ABB RAPID module: P708.mod

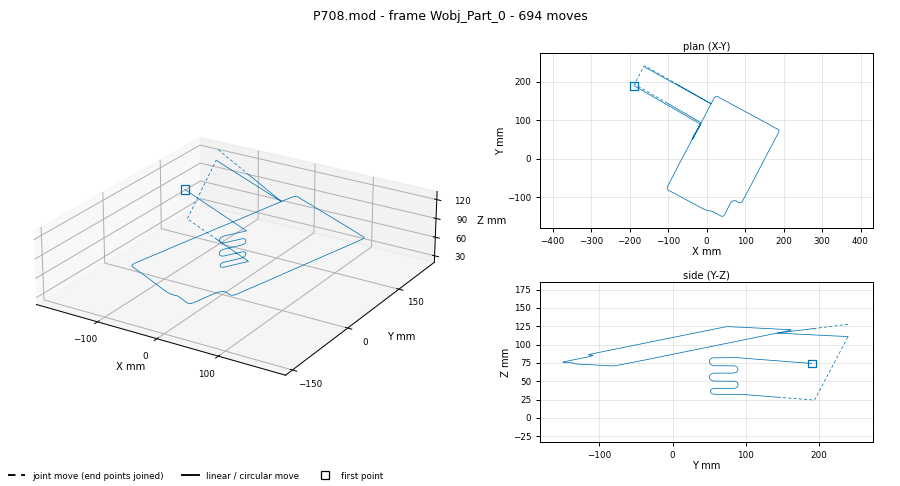
[picture p0: tool path of P708.mod in frame Wobj_Part_0, 694 of 704 moves have a stored position in this frame; points joined in program order, loops and branches not executed]
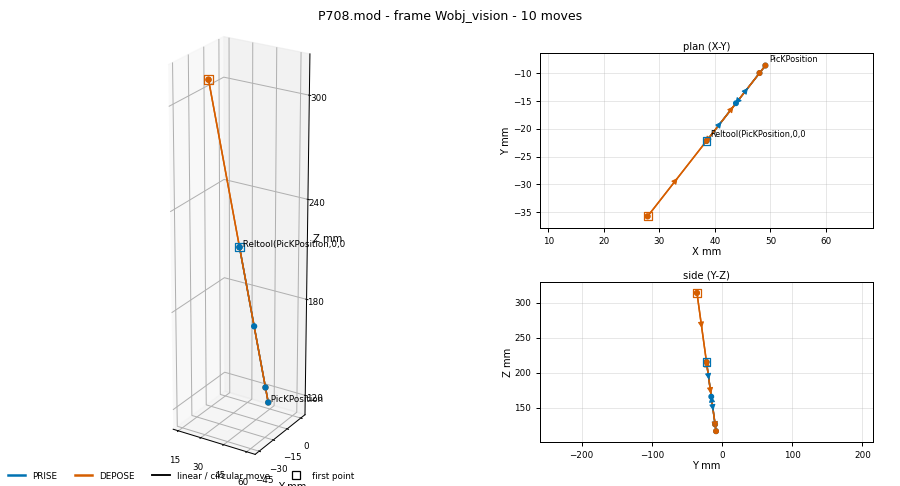
[picture p1: tool path of P708.mod in frame Wobj_vision, 10 of 704 moves have a stored position in this frame; points joined in program order, loops and branches not executed]
MODULE P708

    ! Nom         :P708
    ! Description :
    ! Créé le     :31/05/2023 18:09:45

    LOCAL CONST SPEEDDATA VitesseLente :=[3,500,0,0];
	LOCAL CONST SPEEDDATA VitesseRapide :=[30,500,0,0];
	LOCAL CONST SPEEDDATA VitesseTronconnage :=[2,500,0,0];
	LOCAL CONST SPEEDDATA VitesseTronconnageApp :=[10,500,0,0];
    !
    !Point de prise
    LOCAL PERS Robtarget PicKPosition := [[49.097436543476,-8.59484692597384,116.899947760068],[0.0805571048843757,-0.506621283374927,0.857813762365557,0.0316382234083716],[0,0,0,0],[8.999999E+09,8.999999E+09,8.999999E+09,8.999999E+09,8.999999E+09,8.999999E+09]];
	LOCAL PERS Pose Ref := [[0,0,0],[1,0,0,0]];
    !
    !Declaration des points de meulage

    !Tr_meulage_motif_1 : Meulage d'un motif
    LOCAL CONST Robtarget Tr_meulage_motif_1_0 := [[-15.398982421875,89.8560390625,82.14859375],[0.360190468749215,-0.346276211408762,0.600337290207395,-0.624460366733596],[0,0,0,0],[8.999999E+09,8.999999E+09,8.999999E+09,8.999999E+09,8.999999E+09,8.999999E+09]];
    LOCAL CONST Robtarget Tr_meulage_motif_1_1 := [[-15.875765625,88.977015625,82.148578125],[0.360190468749215,-0.346276211408762,0.600337290207395,-0.624460366733596],[0,0,0,0],[8.999999E+09,8.999999E+09,8.999999E+09,8.999999E+09,8.999999E+09,8.999999E+09]];
    LOCAL CONST Robtarget Tr_meulage_motif_1_2 := [[-16.352548828125,88.0979921875,82.1485625],[0.360190468749215,-0.346276211408762,0.600337290207395,-0.624460366733596],[0,0,0,0],[8.999999E+09,8.999999E+09,8.999999E+09,8.999999E+09,8.999999E+09,8.999999E+09]];
    LOCAL CONST Robtarget Tr_meulage_motif_1_3 := [[-16.82933203125,87.2189765625,82.148546875],[0.360190468749215,-0.346276211408762,0.600337290207395,-0.624460366733596],[0,0,0,0],[8.999999E+09,8.999999E+09,8.999999E+09,8.999999E+09,8.999999E+09,8.999999E+09]];
    LOCAL CONST Robtarget Tr_meulage_motif_1_4 := [[-17.306115234375,86.339953125,82.14853125],[0.360190468749215,-0.346276211408762,0.600337290207395,-0.624460366733596],[0,0,0,0],[8.999999E+09,8.999999E+09,8.999999E+09,8.999999E+09,8.999999E+09,8.999999E+09]];
    LOCAL CONST Robtarget Tr_meulage_motif_1_5 := [[-17.7828984375,85.4609296875,82.1485078125],[0.360190468749215,-0.346276211408762,0.600337290207395,-0.624460366733596],[0,0,0,0],[8.999999E+09,8.999999E+09,8.999999E+09,8.999999E+09,8.999999E+09,8.999999E+09]];
    LOCAL CONST Robtarget Tr_meulage_motif_1_6 := [[-18.259681640625,84.5819140625,82.1484921875],[0.360190468749215,-0.346276211408762,0.600337290207395,-0.624460366733596],[0,0,0,0],[8.999999E+09,8.999999E+09,8.999999E+09,8.999999E+09,8.999999E+09,8.999999E+09]];
    LOCAL CONST Robtarget Tr_meulage_motif_1_7 := [[-18.736462890625,83.702890625,82.1484765625],[0.360190468749215,-0.346276211408762,0.600337290207395,-0.624460366733596],[0,0,0,0],[8.999999E+09,8.999999E+09,8.999999E+09,8.999999E+09,8.999999E+09,8.999999E+09]];
    LOCAL CONST Robtarget Tr_meulage_motif_1_8 := [[-19.21324609375,82.8238671875,82.1484609375],[0.360190468749215,-0.346276211408762,0.600337290207395,-0.624460366733596],[0,0,0,0],[8.999999E+09,8.999999E+09,8.999999E+09,8.999999E+09,8.999999E+09,8.999999E+09]];
    LOCAL CONST Robtarget Tr_meulage_motif_1_9 := [[-19.690029296875,81.9448515625,82.1484453125],[0.360190468749215,-0.346276211408762,0.600337290207395,-0.624460366733596],[0,0,0,0],[8.999999E+09,8.999999E+09,8.999999E+09,8.999999E+09,8.999999E+09,8.999999E+09]];
    LOCAL CONST Robtarget Tr_meulage_motif_1_10 := [[-20.1668125,81.065828125,82.1484296875],[0.360190468749215,-0.346276211408762,0.600337290207395,-0.624460366733596],[0,0,0,0],[8.999999E+09,8.999999E+09,8.999999E+09,8.999999E+09,8.999999E+09,8.999999E+09]];
    LOCAL CONST Robtarget Tr_meulage_motif_1_11 := [[-20.643595703125,80.1868046875,82.1484140625],[0.360190468749215,-0.346276211408762,0.600337290207395,-0.624460366733596],[0,0,0,0],[8.999999E+09,8.999999E+09,8.999999E+09,8.999999E+09,8.999999E+09,8.999999E+09]];
    LOCAL CONST Robtarget Tr_meulage_motif_1_12 := [[-21.12037890625,79.3077890625,82.1483984375],[0.360190468749215,-0.346276211408762,0.600337290207395,-0.624460366733596],[0,0,0,0],[8.999999E+09,8.999999E+09,8.999999E+09,8.999999E+09,8.999999E+09,8.999999E+09]];
    LOCAL CONST Robtarget Tr_meulage_motif_1_13 := [[-21.597162109375,78.428765625,82.1483828125],[0.360190468749215,-0.346276211408762,0.600337290207395,-0.624460366733596],[0,0,0,0],[8.999999E+09,8.999999E+09,8.999999E+09,8.999999E+09,8.999999E+09,8.999999E+09]];
    LOCAL CONST Robtarget Tr_meulage_motif_1_14 := [[-22.0739453125,77.5497421875,82.1483671875],[0.360190468749215,-0.346276211408762,0.600337290207395,-0.624460366733596],[0,0,0,0],[8.999999E+09,8.999999E+09,8.999999E+09,8.999999E+09,8.999999E+09,8.999999E+09]];
    LOCAL CONST Robtarget Tr_meulage_motif_1_15 := [[-22.550728515625,76.6707265625,82.1483515625],[0.360190468749215,-0.346276211408762,0.600337290207395,-0.624460366733596],[0,0,0,0],[8.999999E+09,8.999999E+09,8.999999E+09,8.999999E+09,8.999999E+09,8.999999E+09]];
    LOCAL CONST Robtarget Tr_meulage_motif_1_16 := [[-23.02751171875,75.791703125,82.1483359375],[0.360190468749215,-0.346276211408762,0.600337290207395,-0.624460366733596],[0,0,0,0],[8.999999E+09,8.999999E+09,8.999999E+09,8.999999E+09,8.999999E+09,8.999999E+09]];
    LOCAL CONST Robtarget Tr_meulage_motif_1_17 := [[-23.504294921875,74.9126796875,82.1483203125],[0.360190468749215,-0.346276211408762,0.600337290207395,-0.624460366733596],[0,0,0,0],[8.999999E+09,8.999999E+09,8.999999E+09,8.999999E+09,8.999999E+09,8.999999E+09]];
    LOCAL CONST Robtarget Tr_meulage_motif_1_18 := [[-23.981078125,74.03365625,82.1483046875],[0.360190468749215,-0.346276211408762,0.600337290207395,-0.624460366733596],[0,0,0,0],[8.999999E+09,8.999999E+09,8.999999E+09,8.999999E+09,8.999999E+09,8.999999E+09]];
    LOCAL CONST Robtarget Tr_meulage_motif_1_19 := [[-24.457861328125,73.154640625,82.1482890625],[0.360190468749215,-0.346276211408762,0.600337290207395,-0.624460366733596],[0,0,0,0],[8.999999E+09,8.999999E+09,8.999999E+09,8.999999E+09,8.999999E+09,8.999999E+09]];
    LOCAL CONST Robtarget Tr_meulage_motif_1_20 := [[-24.93464453125,72.2756171875,82.1482734375],[0.360190468749215,-0.346276211408762,0.600337290207395,-0.624460366733596],[0,0,0,0],[8.999999E+09,8.999999E+09,8.999999E+09,8.999999E+09,8.999999E+09,8.999999E+09]];
    LOCAL CONST Robtarget Tr_meulage_motif_1_21 := [[-25.411427734375,71.39659375,82.1482578125],[0.360190468749215,-0.346276211408762,0.600337290207395,-0.624460366733596],[0,0,0,0],[8.999999E+09,8.999999E+09,8.999999E+09,8.999999E+09,8.999999E+09,8.999999E+09]];
    LOCAL CONST Robtarget Tr_meulage_motif_1_22 := [[-25.888208984375,70.517578125,82.1482421875],[0.360190468749215,-0.346276211408762,0.600337290207395,-0.624460366733596],[0,0,0,0],[8.999999E+09,8.999999E+09,8.999999E+09,8.999999E+09,8.999999E+09,8.999999E+09]];
    LOCAL CONST Robtarget Tr_meulage_motif_1_23 := [[-26.3649921875,69.6385546875,82.14821875],[0.360190468749215,-0.346276211408762,0.600337290207395,-0.624460366733596],[0,0,0,0],[8.999999E+09,8.999999E+09,8.999999E+09,8.999999E+09,8.999999E+09,8.999999E+09]];
    LOCAL CONST Robtarget Tr_meulage_motif_1_24 := [[-26.841775390625,68.75953125,82.148203125],[0.360190468749215,-0.346276211408762,0.600337290207395,-0.624460366733596],[0,0,0,0],[8.999999E+09,8.999999E+09,8.999999E+09,8.999999E+09,8.999999E+09,8.999999E+09]];
    LOCAL CONST Robtarget Tr_meulage_motif_1_25 := [[-27.31855859375,67.880515625,82.1481875],[0.360190468749215,-0.346276211408762,0.600337290207395,-0.624460366733596],[0,0,0,0],[8.999999E+09,8.999999E+09,8.999999E+09,8.999999E+09,8.999999E+09,8.999999E+09]];
    LOCAL CONST Robtarget Tr_meulage_motif_1_26 := [[-27.795341796875,67.0014921875,82.148171875],[0.360190468749215,-0.346276211408762,0.600337290207395,-0.624460366733596],[0,0,0,0],[8.999999E+09,8.999999E+09,8.999999E+09,8.999999E+09,8.999999E+09,8.999999E+09]];
    LOCAL CONST Robtarget Tr_meulage_motif_1_27 := [[-28.272125,66.12246875,82.14815625],[0.360190468749215,-0.346276211408762,0.600337290207395,-0.624460366733596],[0,0,0,0],[8.999999E+09,8.999999E+09,8.999999E+09,8.999999E+09,8.999999E+09,8.999999E+09]];
    LOCAL CONST Robtarget Tr_meulage_motif_1_28 := [[-28.748908203125,65.24344921875,82.148140625],[0.360190468749215,-0.346276211408762,0.600337290207395,-0.624460366733596],[0,0,0,0],[8.999999E+09,8.999999E+09,8.999999E+09,8.999999E+09,8.999999E+09,8.999999E+09]];
    LOCAL CONST Robtarget Tr_meulage_motif_1_29 := [[-29.22569140625,64.3644296875,82.148125],[0.360190468749215,-0.346276211408762,0.600337290207395,-0.624460366733596],[0,0,0,0],[8.999999E+09,8.999999E+09,8.999999E+09,8.999999E+09,8.999999E+09,8.999999E+09]];
    LOCAL CONST Robtarget Tr_meulage_motif_1_30 := [[-29.702474609375,63.48540625,82.148109375],[0.360190468749215,-0.346276211408762,0.600337290207395,-0.624460366733596],[0,0,0,0],[8.999999E+09,8.999999E+09,8.999999E+09,8.999999E+09,8.999999E+09,8.999999E+09]];
    LOCAL CONST Robtarget Tr_meulage_motif_1_31 := [[-30.1792578125,62.60638671875,82.14809375],[0.360190468749215,-0.346276211408762,0.600337290207395,-0.624460366733596],[0,0,0,0],[8.999999E+09,8.999999E+09,8.999999E+09,8.999999E+09,8.999999E+09,8.999999E+09]];
    LOCAL CONST Robtarget Tr_meulage_motif_1_32 := [[-30.656041015625,61.7273671875,82.148078125],[0.360190468749215,-0.346276211408762,0.600337290207395,-0.624460366733596],[0,0,0,0],[8.999999E+09,8.999999E+09,8.999999E+09,8.999999E+09,8.999999E+09,8.999999E+09]];
    LOCAL CONST Robtarget Tr_meulage_motif_1_33 := [[-31.13282421875,60.84834375,82.1480625],[0.360190468749215,-0.346276211408762,0.600337290207395,-0.624460366733596],[0,0,0,0],[8.999999E+09,8.999999E+09,8.999999E+09,8.999999E+09,8.999999E+09,8.999999E+09]];
    LOCAL CONST Robtarget Tr_meulage_motif_1_34 := [[-31.609607421875,59.96932421875,82.148046875],[0.360190468749215,-0.346276211408762,0.600337290207395,-0.624460366733596],[0,0,0,0],[8.999999E+09,8.999999E+09,8.999999E+09,8.999999E+09,8.999999E+09,8.999999E+09]];
    LOCAL CONST Robtarget Tr_meulage_motif_1_35 := [[-32.086390625,59.0903046875,82.14803125],[0.360190468749215,-0.346276211408762,0.600337290207395,-0.624460366733596],[0,0,0,0],[8.999999E+09,8.999999E+09,8.999999E+09,8.999999E+09,8.999999E+09,8.999999E+09]];
    LOCAL CONST Robtarget Tr_meulage_motif_1_36 := [[-32.563173828125,58.21128125,82.148015625],[0.360190468749215,-0.346276211408762,0.600337290207395,-0.624460366733596],[0,0,0,0],[8.999999E+09,8.999999E+09,8.999999E+09,8.999999E+09,8.999999E+09,8.999999E+09]];
    LOCAL CONST Robtarget Tr_meulage_motif_1_37 := [[-33.03995703125,57.33226171875,82.148],[0.360190468749215,-0.346276211408762,0.600337290207395,-0.624460366733596],[0,0,0,0],[8.999999E+09,8.999999E+09,8.999999E+09,8.999999E+09,8.999999E+09,8.999999E+09]];
    LOCAL CONST Robtarget Tr_meulage_motif_1_38 := [[-33.51673828125,56.45323828125,82.147984375],[0.360190468749215,-0.346276211408762,0.600337290207395,-0.624460366733596],[0,0,0,0],[8.999999E+09,8.999999E+09,8.999999E+09,8.999999E+09,8.999999E+09,8.999999E+09]];
    LOCAL CONST Robtarget Tr_meulage_motif_1_39 := [[-33.9913828125,55.58151953125,82.0373828125],[0.360190468749215,-0.346276211408762,0.600337290207395,-0.624460366733596],[0,0,0,0],[8.999999E+09,8.999999E+09,8.999999E+09,8.999999E+09,8.999999E+09,8.999999E+09]];
    LOCAL CONST Robtarget Tr_meulage_motif_1_40 := [[-34.44533984375,54.75098828125,81.826203125],[0.360190468749215,-0.346276211408762,0.600337290207395,-0.624460366733596],[0,0,0,0],[8.999999E+09,8.999999E+09,8.999999E+09,8.999999E+09,8.999999E+09,8.999999E+09]];
    LOCAL CONST Robtarget Tr_meulage_motif_1_41 := [[-34.855359375,54.00330859375,81.554375],[0.360190468749215,-0.346276211408762,0.600337290207395,-0.624460366733596],[0,0,0,0],[8.999999E+09,8.999999E+09,8.999999E+09,8.999999E+09,8.999999E+09,8.999999E+09]];
    LOCAL CONST Robtarget Tr_meulage_motif_1_42 := [[-35.216421875,53.34600390625,81.278453125],[0.360190468749215,-0.346276211408762,0.600337290207395,-0.624460366733596],[0,0,0,0],[8.999999E+09,8.999999E+09,8.999999E+09,8.999999E+09,8.999999E+09,8.999999E+09]];
    LOCAL CONST Robtarget Tr_meulage_motif_1_43 := [[-35.74921875,52.38240625,80.662375],[0.360190468749215,-0.346276211408762,0.600337290207395,-0.624460366733596],[0,0,0,0],[8.999999E+09,8.999999E+09,8.999999E+09,8.999999E+09,8.999999E+09,8.999999E+09]];
    LOCAL CONST Robtarget Tr_meulage_motif_1_44 := [[-36.24816015625,51.4882578125,79.8147890625],[0.360190468749215,-0.346276211408762,0.600337290207395,-0.624460366733596],[0,0,0,0],[8.999999E+09,8.999999E+09,8.999999E+09,8.999999E+09,8.999999E+09,8.999999E+09]];
    LOCAL CONST Robtarget Tr_meulage_motif_1_45 := [[-36.6653203125,50.7502265625,78.7910078125],[0.360190468749215,-0.346276211408762,0.600337290207395,-0.624460366733596],[0,0,0,0],[8.999999E+09,8.999999E+09,8.999999E+09,8.999999E+09,8.999999E+09,8.999999E+09]];
    LOCAL CONST Robtarget Tr_meulage_motif_1_46 := [[-36.91225,50.32884375,77.6749296875],[0.360190468749215,-0.346276211408762,0.600337290207395,-0.624460366733596],[0,0,0,0],[8.999999E+09,8.999999E+09,8.999999E+09,8.999999E+09,8.999999E+09,8.999999E+09]];
    LOCAL CONST Robtarget Tr_meulage_motif_1_47 := [[-36.934,50.30986328125,76.97903125],[0.360190468749215,-0.346276211408762,0.600337290207395,-0.624460366733596],[0,0,0,0],[8.999999E+09,8.999999E+09,8.999999E+09,8.999999E+09,8.999999E+09,8.999999E+09]];
    LOCAL CONST Robtarget Tr_meulage_motif_1_48 := [[-36.94240234375,50.31443359375,76.3178515625],[0.360190468749215,-0.346276211408762,0.600337290207395,-0.624460366733596],[0,0,0,0],[8.999999E+09,8.999999E+09,8.999999E+09,8.999999E+09,8.999999E+09,8.999999E+09]];
    LOCAL CONST Robtarget Tr_meulage_motif_1_49 := [[-36.924640625,50.3672421875,75.656828125],[0.360190468749215,-0.346276211408762,0.600337290207395,-0.624460366733596],[0,0,0,0],[8.999999E+09,8.999999E+09,8.999999E+09,8.999999E+09,8.999999E+09,8.999999E+09]];
    LOCAL CONST Robtarget Tr_meulage_motif_1_50 := [[-36.7011015625,50.81280078125,74.555203125],[0.360190468749215,-0.346276211408762,0.600337290207395,-0.624460366733596],[0,0,0,0],[8.999999E+09,8.999999E+09,8.999999E+09,8.999999E+09,8.999999E+09,8.999999E+09]];
    LOCAL CONST Robtarget Tr_meulage_motif_1_51 := [[-36.30547265625,51.57275,73.5486953125],[0.360190468749215,-0.346276211408762,0.600337290207395,-0.624460366733596],[0,0,0,0],[8.999999E+09,8.999999E+09,8.999999E+09,8.999999E+09,8.999999E+09,8.999999E+09]];
    LOCAL CONST Robtarget Tr_meulage_motif_1_52 := [[-35.8280625,52.47807421875,72.7199296875],[0.360190468749215,-0.346276211408762,0.600337290207395,-0.624460366733596],[0,0,0,0],[8.999999E+09,8.999999E+09,8.999999E+09,8.999999E+09,8.999999E+09,8.999999E+09]];
    LOCAL CONST Robtarget Tr_meulage_motif_1_53 := [[-35.5055,53.08477734375,72.3242265625],[0.360190468749215,-0.346276211408762,0.600337290207395,-0.624460366733596],[0,0,0,0],[8.999999E+09,8.999999E+09,8.999999E+09,8.999999E+09,8.999999E+09,8.999999E+09]];
    LOCAL CONST Robtarget Tr_meulage_motif_1_54 := [[-34.95950390625,54.10619140625,71.836765625],[0.360190468749215,-0.346276211408762,0.600337290207395,-0.624460366733596],[0,0,0,0],[8.999999E+09,8.999999E+09,8.999999E+09,8.999999E+09,8.999999E+09,8.999999E+09]];
    LOCAL CONST Robtarget Tr_meulage_motif_1_55 := [[-34.55996484375,54.85081640625,71.5727109375],[0.360190468749215,-0.346276211408762,0.600337290207395,-0.624460366733596],[0,0,0,0],[8.999999E+09,8.999999E+09,8.999999E+09,8.999999E+09,8.999999E+09,8.999999E+09]];
    LOCAL CONST Robtarget Tr_meulage_motif_1_56 := [[-34.118203125,55.67148046875,71.36828125],[0.360190468749215,-0.346276211408762,0.600337290207395,-0.624460366733596],[0,0,0,0],[8.999999E+09,8.999999E+09,8.999999E+09,8.999999E+09,8.999999E+09,8.999999E+09]];
    LOCAL CONST Robtarget Tr_meulage_motif_1_57 := [[-33.65158984375,56.53504296875,71.25971875],[0.360190468749215,-0.346276211408762,0.600337290207395,-0.624460366733596],[0,0,0,0],[8.999999E+09,8.999999E+09,8.999999E+09,8.999999E+09,8.999999E+09,8.999999E+09]];
    LOCAL CONST Robtarget Tr_meulage_motif_1_58 := [[-33.1797578125,57.40829296875,71.1491484375],[0.360190468749215,-0.346276211408762,0.600337290207395,-0.624460366733596],[0,0,0,0],[8.999999E+09,8.999999E+09,8.999999E+09,8.999999E+09,8.999999E+09,8.999999E+09]];
    LOCAL CONST Robtarget Tr_meulage_motif_1_59 := [[-32.702974609375,58.2873125,71.1491640625],[0.360190468749215,-0.346276211408762,0.600337290207395,-0.624460366733596],[0,0,0,0],[8.999999E+09,8.999999E+09,8.999999E+09,8.999999E+09,8.999999E+09,8.999999E+09]];
    LOCAL CONST Robtarget Tr_meulage_motif_1_60 := [[-32.22619140625,59.16633203125,71.1491796875],[0.360190468749215,-0.346276211408762,0.600337290207395,-0.624460366733596],[0,0,0,0],[8.999999E+09,8.999999E+09,8.999999E+09,8.999999E+09,8.999999E+09,8.999999E+09]];
    LOCAL CONST Robtarget Tr_meulage_motif_1_61 := [[-31.74941015625,60.04535546875,71.1491953125],[0.360190468749215,-0.346276211408762,0.600337290207395,-0.624460366733596],[0,0,0,0],[8.999999E+09,8.999999E+09,8.999999E+09,8.999999E+09,8.999999E+09,8.999999E+09]];
    LOCAL CONST Robtarget Tr_meulage_motif_1_62 := [[-31.272626953125,60.924375,71.1492109375],[0.360190468749215,-0.346276211408762,0.600337290207395,-0.624460366733596],[0,0,0,0],[8.999999E+09,8.999999E+09,8.999999E+09,8.999999E+09,8.999999E+09,8.999999E+09]];
    LOCAL CONST Robtarget Tr_meulage_motif_1_63 := [[-30.79584375,61.80339453125,71.1492265625],[0.360190468749215,-0.346276211408762,0.600337290207395,-0.624460366733596],[0,0,0,0],[8.999999E+09,8.999999E+09,8.999999E+09,8.999999E+09,8.999999E+09,8.999999E+09]];
    LOCAL CONST Robtarget Tr_meulage_motif_1_64 := [[-30.319060546875,62.68241796875,71.1492421875],[0.360190468749215,-0.346276211408762,0.600337290207395,-0.624460366733596],[0,0,0,0],[8.999999E+09,8.999999E+09,8.999999E+09,8.999999E+09,8.999999E+09,8.999999E+09]];
    LOCAL CONST Robtarget Tr_meulage_motif_1_65 := [[-29.84227734375,63.5614375,71.1492578125],[0.360190468749215,-0.346276211408762,0.600337290207395,-0.624460366733596],[0,0,0,0],[8.999999E+09,8.999999E+09,8.999999E+09,8.999999E+09,8.999999E+09,8.999999E+09]];
    LOCAL CONST Robtarget Tr_meulage_motif_1_66 := [[-29.365494140625,64.4404609375,71.14928125],[0.360190468749215,-0.346276211408762,0.600337290207395,-0.624460366733596],[0,0,0,0],[8.999999E+09,8.999999E+09,8.999999E+09,8.999999E+09,8.999999E+09,8.999999E+09]];
    LOCAL CONST Robtarget Tr_meulage_motif_1_67 := [[-28.8887109375,65.31948046875,71.149296875],[0.360190468749215,-0.346276211408762,0.600337290207395,-0.624460366733596],[0,0,0,0],[8.999999E+09,8.999999E+09,8.999999E+09,8.999999E+09,8.999999E+09,8.999999E+09]];
    LOCAL CONST Robtarget Tr_meulage_motif_1_68 := [[-28.411927734375,66.1985,71.1493125],[0.360190468749215,-0.346276211408762,0.600337290207395,-0.624460366733596],[0,0,0,0],[8.999999E+09,8.999999E+09,8.999999E+09,8.999999E+09,8.999999E+09,8.999999E+09]];
    LOCAL CONST Robtarget Tr_meulage_motif_1_69 := [[-27.93514453125,67.0775234375,71.149328125],[0.360190468749215,-0.346276211408762,0.600337290207395,-0.624460366733596],[0,0,0,0],[8.999999E+09,8.999999E+09,8.999999E+09,8.999999E+09,8.999999E+09,8.999999E+09]];
    LOCAL CONST Robtarget Tr_meulage_motif_1_70 := [[-27.458361328125,67.956546875,71.14934375],[0.360190468749215,-0.346276211408762,0.600337290207395,-0.624460366733596],[0,0,0,0],[8.999999E+09,8.999999E+09,8.999999E+09,8.999999E+09,8.999999E+09,8.999999E+09]];
    LOCAL CONST Robtarget Tr_meulage_motif_1_71 := [[-26.981578125,68.8355625,71.149359375],[0.360190468749215,-0.346276211408762,0.600337290207395,-0.624460366733596],[0,0,0,0],[8.999999E+09,8.999999E+09,8.999999E+09,8.999999E+09,8.999999E+09,8.999999E+09]];
    LOCAL CONST Robtarget Tr_meulage_motif_1_72 := [[-26.504794921875,69.7145859375,71.149375],[0.360190468749215,-0.346276211408762,0.600337290207395,-0.624460366733596],[0,0,0,0],[8.999999E+09,8.999999E+09,8.999999E+09,8.999999E+09,8.999999E+09,8.999999E+09]];
    LOCAL CONST Robtarget Tr_meulage_motif_1_73 := [[-26.02801171875,70.593609375,71.149390625],[0.360190468749215,-0.346276211408762,0.600337290207395,-0.624460366733596],[0,0,0,0],[8.999999E+09,8.999999E+09,8.999999E+09,8.999999E+09,8.999999E+09,8.999999E+09]];
    LOCAL CONST Robtarget Tr_meulage_motif_1_74 := [[-25.551228515625,71.472625,71.14940625],[0.360190468749215,-0.346276211408762,0.600337290207395,-0.624460366733596],[0,0,0,0],[8.999999E+09,8.999999E+09,8.999999E+09,8.999999E+09,8.999999E+09,8.999999E+09]];
    LOCAL CONST Robtarget Tr_meulage_motif_1_75 := [[-25.0744453125,72.3516484375,71.149421875],[0.360190468749215,-0.346276211408762,0.600337290207395,-0.624460366733596],[0,0,0,0],[8.999999E+09,8.999999E+09,8.999999E+09,8.999999E+09,8.999999E+09,8.999999E+09]];
    LOCAL CONST Robtarget Tr_meulage_motif_1_76 := [[-24.5976640625,73.230671875,71.1494375],[0.360190468749215,-0.346276211408762,0.600337290207395,-0.624460366733596],[0,0,0,0],[8.999999E+09,8.999999E+09,8.999999E+09,8.999999E+09,8.999999E+09,8.999999E+09]];
    LOCAL CONST Robtarget Tr_meulage_motif_1_77 := [[-24.120880859375,74.1096875,71.149453125],[0.360190468749215,-0.346276211408762,0.600337290207395,-0.624460366733596],[0,0,0,0],[8.999999E+09,8.999999E+09,8.999999E+09,8.999999E+09,8.999999E+09,8.999999E+09]];
    LOCAL CONST Robtarget Tr_meulage_motif_1_78 := [[-23.64409765625,74.9887109375,71.14946875],[0.360190468749215,-0.346276211408762,0.600337290207395,-0.624460366733596],[0,0,0,0],[8.999999E+09,8.999999E+09,8.999999E+09,8.999999E+09,8.999999E+09,8.999999E+09]];
    LOCAL CONST Robtarget Tr_meulage_motif_1_79 := [[-23.167314453125,75.867734375,71.149484375],[0.360190468749215,-0.346276211408762,0.600337290207395,-0.624460366733596],[0,0,0,0],[8.999999E+09,8.999999E+09,8.999999E+09,8.999999E+09,8.999999E+09,8.999999E+09]];
    LOCAL CONST Robtarget Tr_meulage_motif_1_80 := [[-22.69053125,76.74675,71.1495],[0.360190468749215,-0.346276211408762,0.600337290207395,-0.624460366733596],[0,0,0,0],[8.999999E+09,8.999999E+09,8.999999E+09,8.999999E+09,8.999999E+09,8.999999E+09]];
    LOCAL CONST Robtarget Tr_meulage_motif_1_81 := [[-22.213748046875,77.6257734375,71.149515625],[0.360190468749215,-0.346276211408762,0.600337290207395,-0.624460366733596],[0,0,0,0],[8.999999E+09,8.999999E+09,8.999999E+09,8.999999E+09,8.999999E+09,8.999999E+09]];
    LOCAL CONST Robtarget Tr_meulage_motif_1_82 := [[-21.73696484375,78.504796875,71.14953125],[0.360190468749215,-0.346276211408762,0.600337290207395,-0.624460366733596],[0,0,0,0],[8.999999E+09,8.999999E+09,8.999999E+09,8.999999E+09,8.999999E+09,8.999999E+09]];
    LOCAL CONST Robtarget Tr_meulage_motif_1_83 := [[-21.260181640625,79.3838125,71.149546875],[0.360190468749215,-0.346276211408762,0.600337290207395,-0.624460366733596],[0,0,0,0],[8.999999E+09,8.999999E+09,8.999999E+09,8.999999E+09,8.999999E+09,8.999999E+09]];
    LOCAL CONST Robtarget Tr_meulage_motif_1_84 := [[-20.7833984375,80.2628359375,71.1495703125],[0.360190468749215,-0.346276211408762,0.600337290207395,-0.624460366733596],[0,0,0,0],[8.999999E+09,8.999999E+09,8.999999E+09,8.999999E+09,8.999999E+09,8.999999E+09]];
    LOCAL CONST Robtarget Tr_meulage_motif_1_85 := [[-20.306615234375,81.141859375,71.1495859375],[0.360190468749215,-0.346276211408762,0.600337290207395,-0.624460366733596],[0,0,0,0],[8.999999E+09,8.999999E+09,8.999999E+09,8.999999E+09,8.999999E+09,8.999999E+09]];
    LOCAL CONST Robtarget Tr_meulage_motif_1_86 := [[-19.82983203125,82.020875,71.1496015625],[0.360190468749215,-0.346276211408762,0.600337290207395,-0.624460366733596],[0,0,0,0],[8.999999E+09,8.999999E+09,8.999999E+09,8.999999E+09,8.999999E+09,8.999999E+09]];
    LOCAL CONST Robtarget Tr_meulage_motif_1_87 := [[-19.353048828125,82.8998984375,71.1496171875],[0.360190468749215,-0.346276211408762,0.600337290207395,-0.624460366733596],[0,0,0,0],[8.999999E+09,8.999999E+09,8.999999E+09,8.999999E+09,8.999999E+09,8.999999E+09]];
    LOCAL CONST Robtarget Tr_meulage_motif_1_88 := [[-18.876265625,83.778921875,71.1496328125],[0.360190468749215,-0.346276211408762,0.600337290207395,-0.624460366733596],[0,0,0,0],[8.999999E+09,8.999999E+09,8.999999E+09,8.999999E+09,8.999999E+09,8.999999E+09]];
    LOCAL CONST Robtarget Tr_meulage_motif_1_89 := [[-18.404435546875,84.652171875,71.0390625],[0.360190468749215,-0.346276211408762,0.600337290207395,-0.624460366733596],[0,0,0,0],[8.999999E+09,8.999999E+09,8.999999E+09,8.999999E+09,8.999999E+09,8.999999E+09]];
    LOCAL CONST Robtarget Tr_meulage_motif_1_90 := [[-17.95584375,85.485625,70.8279140625],[0.360190468749215,-0.346276211408762,0.600337290207395,-0.624460366733596],[0,0,0,0],[8.999999E+09,8.999999E+09,8.999999E+09,8.999999E+09,8.999999E+09,8.999999E+09]];
    LOCAL CONST Robtarget Tr_meulage_motif_1_91 := [[-17.552736328125,86.2370546875,70.556109375],[0.360190468749215,-0.346276211408762,0.600337290207395,-0.624460366733596],[0,0,0,0],[8.999999E+09,8.999999E+09,8.999999E+09,8.999999E+09,8.999999E+09,8.999999E+09]];
    LOCAL CONST Robtarget Tr_meulage_motif_1_92 := [[-17.21737109375,86.8645859375,70.252],[0.360190468749215,-0.346276211408762,0.600337290207395,-0.624460366733596],[0,0,0,0],[8.999999E+09,8.999999E+09,8.999999E+09,8.999999E+09,8.999999E+09,8.999999E+09]];
    LOCAL CONST Robtarget Tr_meulage_motif_1_93 := [[-16.73257421875,87.778484375,69.5895546875],[0.360190468749215,-0.346276211408762,0.600337290207395,-0.624460366733596],[0,0,0,0],[8.999999E+09,8.999999E+09,8.999999E+09,8.999999E+09,8.999999E+09,8.999999E+09]];
    LOCAL CONST Robtarget Tr_meulage_motif_1_94 := [[-16.3140087890625,88.5775390625,68.6877265625],[0.360190468749215,-0.346276211408762,0.600337290207395,-0.624460366733596],[0,0,0,0],[8.999999E+09,8.999999E+09,8.999999E+09,8.999999E+09,8.999999E+09,8.999999E+09]];
    LOCAL CONST Robtarget Tr_meulage_motif_1_95 := [[-16.0722392578125,89.055015625,67.6418125],[0.360190468749215,-0.346276211408762,0.600337290207395,-0.624460366733596],[0,0,0,0],[8.999999E+09,8.999999E+09,8.999999E+09,8.999999E+09,8.999999E+09,8.999999E+09]];
    LOCAL CONST Robtarget Tr_meulage_motif_1_96 := [[-15.99294921875,89.222234375,66.948671875],[0.360190468749215,-0.346276211408762,0.600337290207395,-0.624460366733596],[0,0,0,0],[8.999999E+09,8.999999E+09,8.999999E+09,8.999999E+09,8.999999E+09,8.999999E+09]];
    LOCAL CONST Robtarget Tr_meulage_motif_1_97 := [[-15.9722958984375,89.2836796875,66.17875],[0.360190468749215,-0.346276211408762,0.600337290207395,-0.624460366733596],[0,0,0,0],[8.999999E+09,8.999999E+09,8.999999E+09,8.999999E+09,8.999999E+09,8.999999E+09]];
    LOCAL CONST Robtarget Tr_meulage_motif_1_98 := [[-16.0139951171875,89.23015625,65.40895703125],[0.360190468749215,-0.346276211408762,0.600337290207395,-0.624460366733596],[0,0,0,0],[8.999999E+09,8.999999E+09,8.999999E+09,8.999999E+09,8.999999E+09,8.999999E+09]];
    LOCAL CONST Robtarget Tr_meulage_motif_1_99 := [[-16.228134765625,88.868984375,64.30081640625],[0.360190468749215,-0.346276211408762,0.600337290207395,-0.624460366733596],[0,0,0,0],[8.999999E+09,8.999999E+09,8.999999E+09,8.999999E+09,8.999999E+09,8.999999E+09]];
    LOCAL CONST Robtarget Tr_meulage_motif_1_100 := [[-16.433115234375,88.50884375,63.71518359375],[0.360190468749215,-0.346276211408762,0.600337290207395,-0.624460366733596],[0,0,0,0],[8.999999E+09,8.999999E+09,8.999999E+09,8.999999E+09,8.999999E+09,8.999999E+09]];
    LOCAL CONST Robtarget Tr_meulage_motif_1_101 := [[-16.867357421875,87.7351796875,62.82813671875],[0.360190468749215,-0.346276211408762,0.600337290207395,-0.624460366733596],[0,0,0,0],[8.999999E+09,8.999999E+09,8.999999E+09,8.999999E+09,8.999999E+09,8.999999E+09]];
    LOCAL CONST Robtarget Tr_meulage_motif_1_102 := [[-17.151869140625,87.2232109375,62.41385546875],[0.360190468749215,-0.346276211408762,0.600337290207395,-0.624460366733596],[0,0,0,0],[8.999999E+09,8.999999E+09,8.999999E+09,8.999999E+09,8.999999E+09,8.999999E+09]];
    LOCAL CONST Robtarget Tr_meulage_motif_1_103 := [[-17.69178125,86.2443046875,61.86980078125],[0.360190468749215,-0.346276211408762,0.600337290207395,-0.624460366733596],[0,0,0,0],[8.999999E+09,8.999999E+09,8.999999E+09,8.999999E+09,8.999999E+09,8.999999E+09]];
    LOCAL CONST Robtarget Tr_meulage_motif_1_104 := [[-18.089166015625,85.5206328125,61.5743203125],[0.360190468749215,-0.346276211408762,0.600337290207395,-0.624460366733596],[0,0,0,0],[8.999999E+09,8.999999E+09,8.999999E+09,8.999999E+09,8.999999E+09,8.999999E+09]];
    LOCAL CONST Robtarget Tr_meulage_motif_1_105 := [[-18.536126953125,84.702796875,61.369859375],[0.360190468749215,-0.346276211408762,0.600337290207395,-0.624460366733596],[0,0,0,0],[8.999999E+09,8.999999E+09,8.999999E+09,8.999999E+09,8.999999E+09,8.999999E+09]];
    LOCAL CONST Robtarget Tr_meulage_motif_1_106 := [[-19.0055,83.840734375,61.2612578125],[0.360190468749215,-0.346276211408762,0.600337290207395,-0.624460366733596],[0,0,0,0],[8.999999E+09,8.999999E+09,8.999999E+09,8.999999E+09,8.999999E+09,8.999999E+09]];
    LOCAL CONST Robtarget Tr_meulage_motif_1_107 := [[-19.480142578125,82.969015625,61.15066015625],[0.360190468749215,-0.346276211408762,0.600337290207395,-0.624460366733596],[0,0,0,0],[8.999999E+09,8.999999E+09,8.999999E+09,8.999999E+09,8.999999E+09,8.999999E+09]];
    LOCAL CONST Robtarget Tr_meulage_motif_1_108 := [[-19.95692578125,82.09,61.15064453125],[0.360190468749215,-0.346276211408762,0.600337290207395,-0.624460366733596],[0,0,0,0],[8.999999E+09,8.999999E+09,8.999999E+09,8.999999E+09,8.999999E+09,8.999999E+09]];
    LOCAL CONST Robtarget Tr_meulage_motif_1_109 := [[-20.433708984375,81.2109765625,61.15062890625],[0.360190468749215,-0.346276211408762,0.600337290207395,-0.624460366733596],[0,0,0,0],[8.999999E+09,8.999999E+09,8.999999E+09,8.999999E+09,8.999999E+09,8.999999E+09]];
    LOCAL CONST Robtarget Tr_meulage_motif_1_110 := [[-20.9104921875,80.331953125,61.15061328125],[0.360190468749215,-0.346276211408762,0.600337290207395,-0.624460366733596],[0,0,0,0],[8.999999E+09,8.999999E+09,8.999999E+09,8.999999E+09,8.999999E+09,8.999999E+09]];
    LOCAL CONST Robtarget Tr_meulage_motif_1_111 := [[-21.387275390625,79.4529375,61.15059765625],[0.360190468749215,-0.346276211408762,0.600337290207395,-0.624460366733596],[0,0,0,0],[8.999999E+09,8.999999E+09,8.999999E+09,8.999999E+09,8.999999E+09,8.999999E+09]];
    LOCAL CONST Robtarget Tr_meulage_motif_1_112 := [[-21.86405859375,78.5739140625,61.15058203125],[0.360190468749215,-0.346276211408762,0.600337290207395,-0.624460366733596],[0,0,0,0],[8.999999E+09,8.999999E+09,8.999999E+09,8.999999E+09,8.999999E+09,8.999999E+09]];
    LOCAL CONST Robtarget Tr_meulage_motif_1_113 := [[-22.340841796875,77.694890625,61.15056640625],[0.360190468749215,-0.346276211408762,0.600337290207395,-0.624460366733596],[0,0,0,0],[8.999999E+09,8.999999E+09,8.999999E+09,8.999999E+09,8.999999E+09,8.999999E+09]];
    LOCAL CONST Robtarget Tr_meulage_motif_1_114 := [[-22.817625,76.815875,61.15055078125],[0.360190468749215,-0.346276211408762,0.600337290207395,-0.624460366733596],[0,0,0,0],[8.999999E+09,8.999999E+09,8.999999E+09,8.999999E+09,8.999999E+09,8.999999E+09]];
    LOCAL CONST Robtarget Tr_meulage_motif_1_115 := [[-23.29440625,75.9368515625,61.15053125],[0.360190468749215,-0.346276211408762,0.600337290207395,-0.624460366733596],[0,0,0,0],[8.999999E+09,8.999999E+09,8.999999E+09,8.999999E+09,8.999999E+09,8.999999E+09]];
    LOCAL CONST Robtarget Tr_meulage_motif_1_116 := [[-23.771189453125,75.057828125,61.150515625],[0.360190468749215,-0.346276211408762,0.600337290207395,-0.624460366733596],[0,0,0,0],[8.999999E+09,8.999999E+09,8.999999E+09,8.999999E+09,8.999999E+09,8.999999E+09]];
    LOCAL CONST Robtarget Tr_meulage_motif_1_117 := [[-24.24797265625,74.1788046875,61.1505],[0.360190468749215,-0.346276211408762,0.600337290207395,-0.624460366733596],[0,0,0,0],[8.999999E+09,8.999999E+09,8.999999E+09,8.999999E+09,8.999999E+09,8.999999E+09]];
    LOCAL CONST Robtarget Tr_meulage_motif_1_118 := [[-24.724755859375,73.2997890625,61.150484375],[0.360190468749215,-0.346276211408762,0.600337290207395,-0.624460366733596],[0,0,0,0],[8.999999E+09,8.999999E+09,8.999999E+09,8.999999E+09,8.999999E+09,8.999999E+09]];
    LOCAL CONST Robtarget Tr_meulage_motif_1_119 := [[-25.2015390625,72.420765625,61.15046875],[0.360190468749215,-0.346276211408762,0.600337290207395,-0.624460366733596],[0,0,0,0],[8.999999E+09,8.999999E+09,8.999999E+09,8.999999E+09,8.999999E+09,8.999999E+09]];
    LOCAL CONST Robtarget Tr_meulage_motif_1_120 := [[-25.678322265625,71.5417421875,61.150453125],[0.360190468749215,-0.346276211408762,0.600337290207395,-0.624460366733596],[0,0,0,0],[8.999999E+09,8.999999E+09,8.999999E+09,8.999999E+09,8.999999E+09,8.999999E+09]];
    LOCAL CONST Robtarget Tr_meulage_motif_1_121 := [[-26.15510546875,70.6627265625,61.1504375],[0.360190468749215,-0.346276211408762,0.600337290207395,-0.624460366733596],[0,0,0,0],[8.999999E+09,8.999999E+09,8.999999E+09,8.999999E+09,8.999999E+09,8.999999E+09]];
    LOCAL CONST Robtarget Tr_meulage_motif_1_122 := [[-26.631888671875,69.783703125,61.150421875],[0.360190468749215,-0.346276211408762,0.600337290207395,-0.624460366733596],[0,0,0,0],[8.999999E+09,8.999999E+09,8.999999E+09,8.999999E+09,8.999999E+09,8.999999E+09]];
    LOCAL CONST Robtarget Tr_meulage_motif_1_123 := [[-27.108671875,68.9046796875,61.15040625],[0.360190468749215,-0.346276211408762,0.600337290207395,-0.624460366733596],[0,0,0,0],[8.999999E+09,8.999999E+09,8.999999E+09,8.999999E+09,8.999999E+09,8.999999E+09]];
    LOCAL CONST Robtarget Tr_meulage_motif_1_124 := [[-27.585455078125,68.0256640625,61.15038671875],[0.360190468749215,-0.346276211408762,0.600337290207395,-0.624460366733596],[0,0,0,0],[8.999999E+09,8.999999E+09,8.999999E+09,8.999999E+09,8.999999E+09,8.999999E+09]];
    LOCAL CONST Robtarget Tr_meulage_motif_1_125 := [[-28.06223828125,67.146640625,61.15037109375],[0.360190468749215,-0.346276211408762,0.600337290207395,-0.624460366733596],[0,0,0,0],[8.999999E+09,8.999999E+09,8.999999E+09,8.999999E+09,8.999999E+09,8.999999E+09]];
    LOCAL CONST Robtarget Tr_meulage_motif_1_126 := [[-28.539021484375,66.2676171875,61.15035546875],[0.360190468749215,-0.346276211408762,0.600337290207395,-0.624460366733596],[0,0,0,0],[8.999999E+09,8.999999E+09,8.999999E+09,8.999999E+09,8.999999E+09,8.999999E+09]];
    LOCAL CONST Robtarget Tr_meulage_motif_1_127 := [[-29.0158046875,65.38859765625,61.15033984375],[0.360190468749215,-0.346276211408762,0.600337290207395,-0.624460366733596],[0,0,0,0],[8.999999E+09,8.999999E+09,8.999999E+09,8.999999E+09,8.999999E+09,8.999999E+09]];
    LOCAL CONST Robtarget Tr_meulage_motif_1_128 := [[-29.492587890625,64.509578125,61.15032421875],[0.360190468749215,-0.346276211408762,0.600337290207395,-0.624460366733596],[0,0,0,0],[8.999999E+09,8.999999E+09,8.999999E+09,8.999999E+09,8.999999E+09,8.999999E+09]];
    LOCAL CONST Robtarget Tr_meulage_motif_1_129 := [[-29.96937109375,63.6305546875,61.15030859375],[0.360190468749215,-0.346276211408762,0.600337290207395,-0.624460366733596],[0,0,0,0],[8.999999E+09,8.999999E+09,8.999999E+09,8.999999E+09,8.999999E+09,8.999999E+09]];
    LOCAL CONST Robtarget Tr_meulage_motif_1_130 := [[-30.44615234375,62.75153515625,61.15029296875],[0.360190468749215,-0.346276211408762,0.600337290207395,-0.624460366733596],[0,0,0,0],[8.999999E+09,8.999999E+09,8.999999E+09,8.999999E+09,8.999999E+09,8.999999E+09]];
    LOCAL CONST Robtarget Tr_meulage_motif_1_131 := [[-30.922935546875,61.872515625,61.15027734375],[0.360190468749215,-0.346276211408762,0.600337290207395,-0.624460366733596],[0,0,0,0],[8.999999E+09,8.999999E+09,8.999999E+09,8.999999E+09,8.999999E+09,8.999999E+09]];
    LOCAL CONST Robtarget Tr_meulage_motif_1_132 := [[-31.39971875,60.9934921875,61.15026171875],[0.360190468749215,-0.346276211408762,0.600337290207395,-0.624460366733596],[0,0,0,0],[8.999999E+09,8.999999E+09,8.999999E+09,8.999999E+09,8.999999E+09,8.999999E+09]];
    LOCAL CONST Robtarget Tr_meulage_motif_1_133 := [[-31.876501953125,60.11447265625,61.1502421875],[0.360190468749215,-0.346276211408762,0.600337290207395,-0.624460366733596],[0,0,0,0],[8.999999E+09,8.999999E+09,8.999999E+09,8.999999E+09,8.999999E+09,8.999999E+09]];
    LOCAL CONST Robtarget Tr_meulage_motif_1_134 := [[-32.35328515625,59.235453125,61.1502265625],[0.360190468749215,-0.346276211408762,0.600337290207395,-0.624460366733596],[0,0,0,0],[8.999999E+09,8.999999E+09,8.999999E+09,8.999999E+09,8.999999E+09,8.999999E+09]];
    LOCAL CONST Robtarget Tr_meulage_motif_1_135 := [[-32.8300703125,58.3564296875,61.1502109375],[0.360190468749215,-0.346276211408762,0.600337290207395,-0.624460366733596],[0,0,0,0],[8.999999E+09,8.999999E+09,8.999999E+09,8.999999E+09,8.999999E+09,8.999999E+09]];
    LOCAL CONST Robtarget Tr_meulage_motif_1_136 := [[-33.3068515625,57.47741015625,61.1501953125],[0.360190468749215,-0.346276211408762,0.600337290207395,-0.624460366733596],[0,0,0,0],[8.999999E+09,8.999999E+09,8.999999E+09,8.999999E+09,8.999999E+09,8.999999E+09]];
    LOCAL CONST Robtarget Tr_meulage_motif_1_137 := [[-33.7836328125,56.59838671875,61.1501796875],[0.360190468749215,-0.346276211408762,0.600337290207395,-0.624460366733596],[0,0,0,0],[8.999999E+09,8.999999E+09,8.999999E+09,8.999999E+09,8.999999E+09,8.999999E+09]];
    LOCAL CONST Robtarget Tr_meulage_motif_1_138 := [[-34.25827734375,55.72666796875,61.03958203125],[0.360190468749215,-0.346276211408762,0.600337290207395,-0.624460366733596],[0,0,0,0],[8.999999E+09,8.999999E+09,8.999999E+09,8.999999E+09,8.999999E+09,8.999999E+09]];
    LOCAL CONST Robtarget Tr_meulage_motif_1_139 := [[-34.71223828125,54.89613671875,60.82840234375],[0.360190468749215,-0.346276211408762,0.600337290207395,-0.624460366733596],[0,0,0,0],[8.999999E+09,8.999999E+09,8.999999E+09,8.999999E+09,8.999999E+09,8.999999E+09]];
    LOCAL CONST Robtarget Tr_meulage_motif_1_140 := [[-35.12225390625,54.14845703125,60.5565703125],[0.360190468749215,-0.346276211408762,0.600337290207395,-0.624460366733596],[0,0,0,0],[8.999999E+09,8.999999E+09,8.999999E+09,8.999999E+09,8.999999E+09,8.999999E+09]];
    LOCAL CONST Robtarget Tr_meulage_motif_1_141 := [[-35.48331640625,53.49115234375,60.28065234375],[0.360190468749215,-0.346276211408762,0.600337290207395,-0.624460366733596],[0,0,0,0],[8.999999E+09,8.999999E+09,8.999999E+09,8.999999E+09,8.999999E+09,8.999999E+09]];
    LOCAL CONST Robtarget Tr_meulage_motif_1_142 := [[-36.0161171875,52.5275546875,59.66457421875],[0.360190468749215,-0.346276211408762,0.600337290207395,-0.624460366733596],[0,0,0,0],[8.999999E+09,8.999999E+09,8.999999E+09,8.999999E+09,8.999999E+09,8.999999E+09]];
    LOCAL CONST Robtarget Tr_meulage_motif_1_143 := [[-36.5150546875,51.63340625,58.81698828125],[0.360190468749215,-0.346276211408762,0.600337290207395,-0.624460366733596],[0,0,0,0],[8.999999E+09,8.999999E+09,8.999999E+09,8.999999E+09,8.999999E+09,8.999999E+09]];
    LOCAL CONST Robtarget Tr_meulage_motif_1_144 := [[-36.93221484375,50.895375,57.79320703125],[0.360190468749215,-0.346276211408762,0.600337290207395,-0.624460366733596],[0,0,0,0],[8.999999E+09,8.999999E+09,8.999999E+09,8.999999E+09,8.999999E+09,8.999999E+09]];
    LOCAL CONST Robtarget Tr_meulage_motif_1_145 := [[-37.1791484375,50.4739921875,56.67712890625],[0.360190468749215,-0.346276211408762,0.600337290207395,-0.624460366733596],[0,0,0,0],[8.999999E+09,8.999999E+09,8.999999E+09,8.999999E+09,8.999999E+09,8.999999E+09]];
    LOCAL CONST Robtarget Tr_meulage_motif_1_146 := [[-37.20089453125,50.45501171875,55.981234375],[0.360190468749215,-0.346276211408762,0.600337290207395,-0.624460366733596],[0,0,0,0],[8.999999E+09,8.999999E+09,8.999999E+09,8.999999E+09,8.999999E+09,8.999999E+09]];
    LOCAL CONST Robtarget Tr_meulage_motif_1_147 := [[-37.20930078125,50.45958203125,55.32005078125],[0.360190468749215,-0.346276211408762,0.600337290207395,-0.624460366733596],[0,0,0,0],[8.999999E+09,8.999999E+09,8.999999E+09,8.999999E+09,8.999999E+09,8.999999E+09]];
    LOCAL CONST Robtarget Tr_meulage_motif_1_148 := [[-37.1915390625,50.512390625,54.65902734375],[0.360190468749215,-0.346276211408762,0.600337290207395,-0.624460366733596],[0,0,0,0],[8.999999E+09,8.999999E+09,8.999999E+09,8.999999E+09,8.999999E+09,8.999999E+09]];
    LOCAL CONST Robtarget Tr_meulage_motif_1_149 := [[-36.968,50.95794921875,53.55740234375],[0.360190468749215,-0.346276211408762,0.600337290207395,-0.624460366733596],[0,0,0,0],[8.999999E+09,8.999999E+09,8.999999E+09,8.999999E+09,8.999999E+09,8.999999E+09]];
    LOCAL CONST Robtarget Tr_meulage_motif_1_150 := [[-36.5723671875,51.7178984375,52.55089453125],[0.360190468749215,-0.346276211408762,0.600337290207395,-0.624460366733596],[0,0,0,0],[8.999999E+09,8.999999E+09,8.999999E+09,8.999999E+09,8.999999E+09,8.999999E+09]];
    LOCAL CONST Robtarget Tr_meulage_motif_1_151 := [[-36.0949609375,52.62322265625,51.722125],[0.360190468749215,-0.346276211408762,0.600337290207395,-0.624460366733596],[0,0,0,0],[8.999999E+09,8.999999E+09,8.999999E+09,8.999999E+09,8.999999E+09,8.999999E+09]];
    LOCAL CONST Robtarget Tr_meulage_motif_1_152 := [[-35.77239453125,53.22992578125,51.32642578125],[0.360190468749215,-0.346276211408762,0.600337290207395,-0.624460366733596],[0,0,0,0],[8.999999E+09,8.999999E+09,8.999999E+09,8.999999E+09,8.999999E+09,8.999999E+09]];
    LOCAL CONST Robtarget Tr_meulage_motif_1_153 := [[-35.22640234375,54.25133984375,50.83896484375],[0.360190468749215,-0.346276211408762,0.600337290207395,-0.624460366733596],[0,0,0,0],[8.999999E+09,8.999999E+09,8.999999E+09,8.999999E+09,8.999999E+09,8.999999E+09]];
    LOCAL CONST Robtarget Tr_meulage_motif_1_154 := [[-34.826859375,54.99596484375,50.57491015625],[0.360190468749215,-0.346276211408762,0.600337290207395,-0.624460366733596],[0,0,0,0],[8.999999E+09,8.999999E+09,8.999999E+09,8.999999E+09,8.999999E+09,8.999999E+09]];
    LOCAL CONST Robtarget Tr_meulage_motif_1_155 := [[-34.38509765625,55.81662890625,50.37048046875],[0.360190468749215,-0.346276211408762,0.600337290207395,-0.624460366733596],[0,0,0,0],[8.999999E+09,8.999999E+09,8.999999E+09,8.999999E+09,8.999999E+09,8.999999E+09]];
    LOCAL CONST Robtarget Tr_meulage_motif_1_156 := [[-33.918484375,56.68019140625,50.2619140625],[0.360190468749215,-0.346276211408762,0.600337290207395,-0.624460366733596],[0,0,0,0],[8.999999E+09,8.999999E+09,8.999999E+09,8.999999E+09,8.999999E+09,8.999999E+09]];
    LOCAL CONST Robtarget Tr_meulage_motif_1_157 := [[-33.44665234375,57.55344140625,50.15134765625],[0.360190468749215,-0.346276211408762,0.600337290207395,-0.624460366733596],[0,0,0,0],[8.999999E+09,8.999999E+09,8.999999E+09,8.999999E+09,8.999999E+09,8.999999E+09]];
    LOCAL CONST Robtarget Tr_meulage_motif_1_158 := [[-32.96987109375,58.4324609375,50.15136328125],[0.360190468749215,-0.346276211408762,0.600337290207395,-0.624460366733596],[0,0,0,0],[8.999999E+09,8.999999E+09,8.999999E+09,8.999999E+09,8.999999E+09,8.999999E+09]];
    LOCAL CONST Robtarget Tr_meulage_motif_1_159 := [[-32.493087890625,59.31148046875,50.15137890625],[0.360190468749215,-0.346276211408762,0.600337290207395,-0.624460366733596],[0,0,0,0],[8.999999E+09,8.999999E+09,8.999999E+09,8.999999E+09,8.999999E+09,8.999999E+09]];
    LOCAL CONST Robtarget Tr_meulage_motif_1_160 := [[-32.0163046875,60.19050390625,50.15139453125],[0.360190468749215,-0.346276211408762,0.600337290207395,-0.624460366733596],[0,0,0,0],[8.999999E+09,8.999999E+09,8.999999E+09,8.999999E+09,8.999999E+09,8.999999E+09]];
    LOCAL CONST Robtarget Tr_meulage_motif_1_161 := [[-31.539521484375,61.0695234375,50.15141015625],[0.360190468749215,-0.346276211408762,0.600337290207395,-0.624460366733596],[0,0,0,0],[8.999999E+09,8.999999E+09,8.999999E+09,8.999999E+09,8.999999E+09,8.999999E+09]];
    LOCAL CONST Robtarget Tr_meulage_motif_1_162 := [[-31.06273828125,61.94854296875,50.15142578125],[0.360190468749215,-0.346276211408762,0.600337290207395,-0.624460366733596],[0,0,0,0],[8.999999E+09,8.999999E+09,8.999999E+09,8.999999E+09,8.999999E+09,8.999999E+09]];
    LOCAL CONST Robtarget Tr_meulage_motif_1_163 := [[-30.585955078125,62.82756640625,50.15144140625],[0.360190468749215,-0.346276211408762,0.600337290207395,-0.624460366733596],[0,0,0,0],[8.999999E+09,8.999999E+09,8.999999E+09,8.999999E+09,8.999999E+09,8.999999E+09]];
    LOCAL CONST Robtarget Tr_meulage_motif_1_164 := [[-30.109171875,63.7065859375,50.1514609375],[0.360190468749215,-0.346276211408762,0.600337290207395,-0.624460366733596],[0,0,0,0],[8.999999E+09,8.999999E+09,8.999999E+09,8.999999E+09,8.999999E+09,8.999999E+09]];
    LOCAL CONST Robtarget Tr_meulage_motif_1_165 := [[-29.632388671875,64.585609375,50.1514765625],[0.360190468749215,-0.346276211408762,0.600337290207395,-0.624460366733596],[0,0,0,0],[8.999999E+09,8.999999E+09,8.999999E+09,8.999999E+09,8.999999E+09,8.999999E+09]];
    LOCAL CONST Robtarget Tr_meulage_motif_1_166 := [[-29.155607421875,65.46462890625,50.1514921875],[0.360190468749215,-0.346276211408762,0.600337290207395,-0.624460366733596],[0,0,0,0],[8.999999E+09,8.999999E+09,8.999999E+09,8.999999E+09,8.999999E+09,8.999999E+09]];
    LOCAL CONST Robtarget Tr_meulage_motif_1_167 := [[-28.67882421875,66.3436484375,50.1515078125],[0.360190468749215,-0.346276211408762,0.600337290207395,-0.624460366733596],[0,0,0,0],[8.999999E+09,8.999999E+09,8.999999E+09,8.999999E+09,8.999999E+09,8.999999E+09]];
    LOCAL CONST Robtarget Tr_meulage_motif_1_168 := [[-28.202041015625,67.222671875,50.1515234375],[0.360190468749215,-0.346276211408762,0.600337290207395,-0.624460366733596],[0,0,0,0],[8.999999E+09,8.999999E+09,8.999999E+09,8.999999E+09,8.999999E+09,8.999999E+09]];
    LOCAL CONST Robtarget Tr_meulage_motif_1_169 := [[-27.7252578125,68.1016953125,50.1515390625],[0.360190468749215,-0.346276211408762,0.600337290207395,-0.624460366733596],[0,0,0,0],[8.999999E+09,8.999999E+09,8.999999E+09,8.999999E+09,8.999999E+09,8.999999E+09]];
    LOCAL CONST Robtarget Tr_meulage_motif_1_170 := [[-27.248474609375,68.9807109375,50.1515546875],[0.360190468749215,-0.346276211408762,0.600337290207395,-0.624460366733596],[0,0,0,0],[8.999999E+09,8.999999E+09,8.999999E+09,8.999999E+09,8.999999E+09,8.999999E+09]];
    LOCAL CONST Robtarget Tr_meulage_motif_1_171 := [[-26.77169140625,69.859734375,50.1515703125],[0.360190468749215,-0.346276211408762,0.600337290207395,-0.624460366733596],[0,0,0,0],[8.999999E+09,8.999999E+09,8.999999E+09,8.999999E+09,8.999999E+09,8.999999E+09]];
    LOCAL CONST Robtarget Tr_meulage_motif_1_172 := [[-26.294908203125,70.7387578125,50.1515859375],[0.360190468749215,-0.346276211408762,0.600337290207395,-0.624460366733596],[0,0,0,0],[8.999999E+09,8.999999E+09,8.999999E+09,8.999999E+09,8.999999E+09,8.999999E+09]];
    LOCAL CONST Robtarget Tr_meulage_motif_1_173 := [[-25.818125,71.6177734375,50.15160546875],[0.360190468749215,-0.346276211408762,0.600337290207395,-0.624460366733596],[0,0,0,0],[8.999999E+09,8.999999E+09,8.999999E+09,8.999999E+09,8.999999E+09,8.999999E+09]];
    LOCAL CONST Robtarget Tr_meulage_motif_1_174 := [[-25.341341796875,72.496796875,50.15162109375],[0.360190468749215,-0.346276211408762,0.600337290207395,-0.624460366733596],[0,0,0,0],[8.999999E+09,8.999999E+09,8.999999E+09,8.999999E+09,8.999999E+09,8.999999E+09]];
    LOCAL CONST Robtarget Tr_meulage_motif_1_175 := [[-24.86455859375,73.3758203125,50.15163671875],[0.360190468749215,-0.346276211408762,0.600337290207395,-0.624460366733596],[0,0,0,0],[8.999999E+09,8.999999E+09,8.999999E+09,8.999999E+09,8.999999E+09,8.999999E+09]];
    LOCAL CONST Robtarget Tr_meulage_motif_1_176 := [[-24.387775390625,74.2548359375,50.15165234375],[0.360190468749215,-0.346276211408762,0.600337290207395,-0.624460366733596],[0,0,0,0],[8.999999E+09,8.999999E+09,8.999999E+09,8.999999E+09,8.999999E+09,8.999999E+09]];
    LOCAL CONST Robtarget Tr_meulage_motif_1_177 := [[-23.9109921875,75.133859375,50.15166796875],[0.360190468749215,-0.346276211408762,0.600337290207395,-0.624460366733596],[0,0,0,0],[8.999999E+09,8.999999E+09,8.999999E+09,8.999999E+09,8.999999E+09,8.999999E+09]];
    LOCAL CONST Robtarget Tr_meulage_motif_1_178 := [[-23.434208984375,76.0128828125,50.15168359375],[0.360190468749215,-0.346276211408762,0.600337290207395,-0.624460366733596],[0,0,0,0],[8.999999E+09,8.999999E+09,8.999999E+09,8.999999E+09,8.999999E+09,8.999999E+09]];
    LOCAL CONST Robtarget Tr_meulage_motif_1_179 := [[-22.95742578125,76.8918984375,50.15169921875],[0.360190468749215,-0.346276211408762,0.600337290207395,-0.624460366733596],[0,0,0,0],[8.999999E+09,8.999999E+09,8.999999E+09,8.999999E+09,8.999999E+09,8.999999E+09]];
    LOCAL CONST Robtarget Tr_meulage_motif_1_180 := [[-22.480642578125,77.770921875,50.15171484375],[0.360190468749215,-0.346276211408762,0.600337290207395,-0.624460366733596],[0,0,0,0],[8.999999E+09,8.999999E+09,8.999999E+09,8.999999E+09,8.999999E+09,8.999999E+09]];
    LOCAL CONST Robtarget Tr_meulage_motif_1_181 := [[-22.003861328125,78.6499453125,50.15173046875],[0.360190468749215,-0.346276211408762,0.600337290207395,-0.624460366733596],[0,0,0,0],[8.999999E+09,8.999999E+09,8.999999E+09,8.999999E+09,8.999999E+09,8.999999E+09]];
    LOCAL CONST Robtarget Tr_meulage_motif_1_182 := [[-21.527078125,79.5289609375,50.15175],[0.360190468749215,-0.346276211408762,0.600337290207395,-0.624460366733596],[0,0,0,0],[8.999999E+09,8.999999E+09,8.999999E+09,8.999999E+09,8.999999E+09,8.999999E+09]];
    LOCAL CONST Robtarget Tr_meulage_motif_1_183 := [[-21.050294921875,80.407984375,50.151765625],[0.360190468749215,-0.346276211408762,0.600337290207395,-0.624460366733596],[0,0,0,0],[8.999999E+09,8.999999E+09,8.999999E+09,8.999999E+09,8.999999E+09,8.999999E+09]];
    LOCAL CONST Robtarget Tr_meulage_motif_1_184 := [[-20.57351171875,81.2870078125,50.15178125],[0.360190468749215,-0.346276211408762,0.600337290207395,-0.624460366733596],[0,0,0,0],[8.999999E+09,8.999999E+09,8.999999E+09,8.999999E+09,8.999999E+09,8.999999E+09]];
    LOCAL CONST Robtarget Tr_meulage_motif_1_185 := [[-20.096728515625,82.1660234375,50.151796875],[0.360190468749215,-0.346276211408762,0.600337290207395,-0.624460366733596],[0,0,0,0],[8.999999E+09,8.999999E+09,8.999999E+09,8.999999E+09,8.999999E+09,8.999999E+09]];
    LOCAL CONST Robtarget Tr_meulage_motif_1_186 := [[-19.6199453125,83.045046875,50.1518125],[0.360190468749215,-0.346276211408762,0.600337290207395,-0.624460366733596],[0,0,0,0],[8.999999E+09,8.999999E+09,8.999999E+09,8.999999E+09,8.999999E+09,8.999999E+09]];
    LOCAL CONST Robtarget Tr_meulage_motif_1_187 := [[-19.143162109375,83.9240703125,50.151828125],[0.360190468749215,-0.346276211408762,0.600337290207395,-0.624460366733596],[0,0,0,0],[8.999999E+09,8.999999E+09,8.999999E+09,8.999999E+09,8.999999E+09,8.999999E+09]];
    LOCAL CONST Robtarget Tr_meulage_motif_1_188 := [[-18.671330078125,84.7973203125,50.04126171875],[0.360190468749215,-0.346276211408762,0.600337290207395,-0.624460366733596],[0,0,0,0],[8.999999E+09,8.999999E+09,8.999999E+09,8.999999E+09,8.999999E+09,8.999999E+09]];
    LOCAL CONST Robtarget Tr_meulage_motif_1_189 := [[-18.222740234375,85.6307734375,49.83011328125],[0.360190468749215,-0.346276211408762,0.600337290207395,-0.624460366733596],[0,0,0,0],[8.999999E+09,8.999999E+09,8.999999E+09,8.999999E+09,8.999999E+09,8.999999E+09]];
    LOCAL CONST Robtarget Tr_meulage_motif_1_190 := [[-17.8196328125,86.382203125,49.55830859375],[0.360190468749215,-0.346276211408762,0.600337290207395,-0.624460366733596],[0,0,0,0],[8.999999E+09,8.999999E+09,8.999999E+09,8.999999E+09,8.999999E+09,8.999999E+09]];
    LOCAL CONST Robtarget Tr_meulage_motif_1_191 := [[-17.484267578125,87.009734375,49.25421484375],[0.360190468749215,-0.346276211408762,0.600337290207395,-0.624460366733596],[0,0,0,0],[8.999999E+09,8.999999E+09,8.999999E+09,8.999999E+09,8.999999E+09,8.999999E+09]];
    LOCAL CONST Robtarget Tr_meulage_motif_1_192 := [[-16.999470703125,87.9236328125,48.59176953125],[0.360190468749215,-0.346276211408762,0.600337290207395,-0.624460366733596],[0,0,0,0],[8.999999E+09,8.999999E+09,8.999999E+09,8.999999E+09,8.999999E+09,8.999999E+09]];
    LOCAL CONST Robtarget Tr_meulage_motif_1_193 := [[-16.580904296875,88.7226875,47.689921875],[0.360190468749215,-0.346276211408762,0.600337290207395,-0.624460366733596],[0,0,0,0],[8.999999E+09,8.999999E+09,8.999999E+09,8.999999E+09,8.999999E+09,8.999999E+09]];
    LOCAL CONST Robtarget Tr_meulage_motif_1_194 := [[-16.339134765625,89.2001640625,46.64402734375],[0.360190468749215,-0.346276211408762,0.600337290207395,-0.624460366733596],[0,0,0,0],[8.999999E+09,8.999999E+09,8.999999E+09,8.999999E+09,8.999999E+09,8.999999E+09]];
    LOCAL CONST Robtarget Tr_meulage_motif_1_195 := [[-16.2598447265625,89.3673828125,45.9508671875],[0.360190468749215,-0.346276211408762,0.600337290207395,-0.624460366733596],[0,0,0,0],[8.999999E+09,8.999999E+09,8.999999E+09,8.999999E+09,8.999999E+09,8.999999E+09]];
    LOCAL CONST Robtarget Tr_meulage_motif_1_196 := [[-16.23919140625,89.428828125,45.18094921875],[0.360190468749215,-0.346276211408762,0.600337290207395,-0.624460366733596],[0,0,0,0],[8.999999E+09,8.999999E+09,8.999999E+09,8.999999E+09,8.999999E+09,8.999999E+09]];
    LOCAL CONST Robtarget Tr_meulage_motif_1_197 := [[-16.280890625,89.3753046875,44.41116796875],[0.360190468749215,-0.346276211408762,0.600337290207395,-0.624460366733596],[0,0,0,0],[8.999999E+09,8.999999E+09,8.999999E+09,8.999999E+09,8.999999E+09,8.999999E+09]];
    LOCAL CONST Robtarget Tr_meulage_motif_1_198 := [[-16.49503125,89.0141328125,43.30302734375],[0.360190468749215,-0.346276211408762,0.600337290207395,-0.624460366733596],[0,0,0,0],[8.999999E+09,8.999999E+09,8.999999E+09,8.999999E+09,8.999999E+09,8.999999E+09]];
    LOCAL CONST Robtarget Tr_meulage_motif_1_199 := [[-16.70001171875,88.6539921875,42.71739453125],[0.360190468749215,-0.346276211408762,0.600337290207395,-0.624460366733596],[0,0,0,0],[8.999999E+09,8.999999E+09,8.999999E+09,8.999999E+09,8.999999E+09,8.999999E+09]];
    LOCAL CONST Robtarget Tr_meulage_motif_1_200 := [[-17.134251953125,87.880328125,41.83031640625],[0.360190468749215,-0.346276211408762,0.600337290207395,-0.624460366733596],[0,0,0,0],[8.999999E+09,8.999999E+09,8.999999E+09,8.999999E+09,8.999999E+09,8.999999E+09]];
    LOCAL CONST Robtarget Tr_meulage_motif_1_201 := [[-17.418763671875,87.368359375,41.4160703125],[0.360190468749215,-0.346276211408762,0.600337290207395,-0.624460366733596],[0,0,0,0],[8.999999E+09,8.999999E+09,8.999999E+09,8.999999E+09,8.999999E+09,8.999999E+09]];
    LOCAL CONST Robtarget Tr_meulage_motif_1_202 := [[-17.958677734375,86.389453125,40.871984375],[0.360190468749215,-0.346276211408762,0.600337290207395,-0.624460366733596],[0,0,0,0],[8.999999E+09,8.999999E+09,8.999999E+09,8.999999E+09,8.999999E+09,8.999999E+09]];
    LOCAL CONST Robtarget Tr_meulage_motif_1_203 := [[-18.3560625,85.66578125,40.57650390625],[0.360190468749215,-0.346276211408762,0.600337290207395,-0.624460366733596],[0,0,0,0],[8.999999E+09,8.999999E+09,8.999999E+09,8.999999E+09,8.999999E+09,8.999999E+09]];
    LOCAL CONST Robtarget Tr_meulage_motif_1_204 := [[-18.8030234375,84.8479453125,40.3720234375],[0.360190468749215,-0.346276211408762,0.600337290207395,-0.624460366733596],[0,0,0,0],[8.999999E+09,8.999999E+09,8.999999E+09,8.999999E+09,8.999999E+09,8.999999E+09]];
    LOCAL CONST Robtarget Tr_meulage_motif_1_205 := [[-19.27239453125,83.9858828125,40.26347265625],[0.360190468749215,-0.346276211408762,0.600337290207395,-0.624460366733596],[0,0,0,0],[8.999999E+09,8.999999E+09,8.999999E+09,8.999999E+09,8.999999E+09,8.999999E+09]];
    LOCAL CONST Robtarget Tr_meulage_motif_1_206 := [[-19.7470390625,83.1141640625,40.152859375],[0.360190468749215,-0.346276211408762,0.600337290207395,-0.624460366733596],[0,0,0,0],[8.999999E+09,8.999999E+09,8.999999E+09,8.999999E+09,8.999999E+09,8.999999E+09]];
    LOCAL CONST Robtarget Tr_meulage_motif_1_207 := [[-20.2238203125,82.2351484375,40.15284375],[0.360190468749215,-0.346276211408762,0.600337290207395,-0.624460366733596],[0,0,0,0],[8.999999E+09,8.999999E+09,8.999999E+09,8.999999E+09,8.999999E+09,8.999999E+09]];
    LOCAL CONST Robtarget Tr_meulage_motif_1_208 := [[-20.700603515625,81.356125,40.152828125],[0.360190468749215,-0.346276211408762,0.600337290207395,-0.624460366733596],[0,0,0,0],[8.999999E+09,8.999999E+09,8.999999E+09,8.999999E+09,8.999999E+09,8.999999E+09]];
    LOCAL CONST Robtarget Tr_meulage_motif_1_209 := [[-21.17738671875,80.4771015625,40.1528125],[0.360190468749215,-0.346276211408762,0.600337290207395,-0.624460366733596],[0,0,0,0],[8.999999E+09,8.999999E+09,8.999999E+09,8.999999E+09,8.999999E+09,8.999999E+09]];
    LOCAL CONST Robtarget Tr_meulage_motif_1_210 := [[-21.654169921875,79.5980859375,40.15279296875],[0.360190468749215,-0.346276211408762,0.600337290207395,-0.624460366733596],[0,0,0,0],[8.999999E+09,8.999999E+09,8.999999E+09,8.999999E+09,8.999999E+09,8.999999E+09]];
    LOCAL CONST Robtarget Tr_meulage_motif_1_211 := [[-22.130953125,78.7190625,40.15277734375],[0.360190468749215,-0.346276211408762,0.600337290207395,-0.624460366733596],[0,0,0,0],[8.999999E+09,8.999999E+09,8.999999E+09,8.999999E+09,8.999999E+09,8.999999E+09]];
    LOCAL CONST Robtarget Tr_meulage_motif_1_212 := [[-22.607736328125,77.8400390625,40.15276171875],[0.360190468749215,-0.346276211408762,0.600337290207395,-0.624460366733596],[0,0,0,0],[8.999999E+09,8.999999E+09,8.999999E+09,8.999999E+09,8.999999E+09,8.999999E+09]];
    LOCAL CONST Robtarget Tr_meulage_motif_1_213 := [[-23.08451953125,76.9610234375,40.15274609375],[0.360190468749215,-0.346276211408762,0.600337290207395,-0.624460366733596],[0,0,0,0],[8.999999E+09,8.999999E+09,8.999999E+09,8.999999E+09,8.999999E+09,8.999999E+09]];
    LOCAL CONST Robtarget Tr_meulage_motif_1_214 := [[-23.561302734375,76.082,40.15273046875],[0.360190468749215,-0.346276211408762,0.600337290207395,-0.624460366733596],[0,0,0,0],[8.999999E+09,8.999999E+09,8.999999E+09,8.999999E+09,8.999999E+09,8.999999E+09]];
    LOCAL CONST Robtarget Tr_meulage_motif_1_215 := [[-24.0380859375,75.2029765625,40.15271484375],[0.360190468749215,-0.346276211408762,0.600337290207395,-0.624460366733596],[0,0,0,0],[8.999999E+09,8.999999E+09,8.999999E+09,8.999999E+09,8.999999E+09,8.999999E+09]];
    LOCAL CONST Robtarget Tr_meulage_motif_1_216 := [[-24.514869140625,74.323953125,40.15269921875],[0.360190468749215,-0.346276211408762,0.600337290207395,-0.624460366733596],[0,0,0,0],[8.999999E+09,8.999999E+09,8.999999E+09,8.999999E+09,8.999999E+09,8.999999E+09]];
    LOCAL CONST Robtarget Tr_meulage_motif_1_217 := [[-24.99165234375,73.4449375,40.15268359375],[0.360190468749215,-0.346276211408762,0.600337290207395,-0.624460366733596],[0,0,0,0],[8.999999E+09,8.999999E+09,8.999999E+09,8.999999E+09,8.999999E+09,8.999999E+09]];
    LOCAL CONST Robtarget Tr_meulage_motif_1_218 := [[-25.468435546875,72.5659140625,40.15266796875],[0.360190468749215,-0.346276211408762,0.600337290207395,-0.624460366733596],[0,0,0,0],[8.999999E+09,8.999999E+09,8.999999E+09,8.999999E+09,8.999999E+09,8.999999E+09]];
    LOCAL CONST Robtarget Tr_meulage_motif_1_219 := [[-25.94521875,71.686890625,40.1526484375],[0.360190468749215,-0.346276211408762,0.600337290207395,-0.624460366733596],[0,0,0,0],[8.999999E+09,8.999999E+09,8.999999E+09,8.999999E+09,8.999999E+09,8.999999E+09]];
    LOCAL CONST Robtarget Tr_meulage_motif_1_220 := [[-26.422001953125,70.807875,40.1526328125],[0.360190468749215,-0.346276211408762,0.600337290207395,-0.624460366733596],[0,0,0,0],[8.999999E+09,8.999999E+09,8.999999E+09,8.999999E+09,8.999999E+09,8.999999E+09]];
    LOCAL CONST Robtarget Tr_meulage_motif_1_221 := [[-26.89878515625,69.9288515625,40.1526171875],[0.360190468749215,-0.346276211408762,0.600337290207395,-0.624460366733596],[0,0,0,0],[8.999999E+09,8.999999E+09,8.999999E+09,8.999999E+09,8.999999E+09,8.999999E+09]];
    LOCAL CONST Robtarget Tr_meulage_motif_1_222 := [[-27.375568359375,69.049828125,40.1526015625],[0.360190468749215,-0.346276211408762,0.600337290207395,-0.624460366733596],[0,0,0,0],[8.999999E+09,8.999999E+09,8.999999E+09,8.999999E+09,8.999999E+09,8.999999E+09]];
    LOCAL CONST Robtarget Tr_meulage_motif_1_223 := [[-27.852349609375,68.1708125,40.1525859375],[0.360190468749215,-0.346276211408762,0.600337290207395,-0.624460366733596],[0,0,0,0],[8.999999E+09,8.999999E+09,8.999999E+09,8.999999E+09,8.999999E+09,8.999999E+09]];
    LOCAL CONST Robtarget Tr_meulage_motif_1_224 := [[-28.3291328125,67.2917890625,40.1525703125],[0.360190468749215,-0.346276211408762,0.600337290207395,-0.624460366733596],[0,0,0,0],[8.999999E+09,8.999999E+09,8.999999E+09,8.999999E+09,8.999999E+09,8.999999E+09]];
    LOCAL CONST Robtarget Tr_meulage_motif_1_225 := [[-28.805916015625,66.412765625,40.1525546875],[0.360190468749215,-0.346276211408762,0.600337290207395,-0.624460366733596],[0,0,0,0],[8.999999E+09,8.999999E+09,8.999999E+09,8.999999E+09,8.999999E+09,8.999999E+09]];
    LOCAL CONST Robtarget Tr_meulage_motif_1_226 := [[-29.28269921875,65.53374609375,40.1525390625],[0.360190468749215,-0.346276211408762,0.600337290207395,-0.624460366733596],[0,0,0,0],[8.999999E+09,8.999999E+09,8.999999E+09,8.999999E+09,8.999999E+09,8.999999E+09]];
    LOCAL CONST Robtarget Tr_meulage_motif_1_227 := [[-29.759482421875,64.6547265625,40.1525234375],[0.360190468749215,-0.346276211408762,0.600337290207395,-0.624460366733596],[0,0,0,0],[8.999999E+09,8.999999E+09,8.999999E+09,8.999999E+09,8.999999E+09,8.999999E+09]];
    LOCAL CONST Robtarget Tr_meulage_motif_1_228 := [[-30.236265625,63.775703125,40.15250390625],[0.360190468749215,-0.346276211408762,0.600337290207395,-0.624460366733596],[0,0,0,0],[8.999999E+09,8.999999E+09,8.999999E+09,8.999999E+09,8.999999E+09,8.999999E+09]];
    LOCAL CONST Robtarget Tr_meulage_motif_1_229 := [[-30.713048828125,62.89668359375,40.15248828125],[0.360190468749215,-0.346276211408762,0.600337290207395,-0.624460366733596],[0,0,0,0],[8.999999E+09,8.999999E+09,8.999999E+09,8.999999E+09,8.999999E+09,8.999999E+09]];
    LOCAL CONST Robtarget Tr_meulage_motif_1_230 := [[-31.18983203125,62.0176640625,40.15247265625],[0.360190468749215,-0.346276211408762,0.600337290207395,-0.624460366733596],[0,0,0,0],[8.999999E+09,8.999999E+09,8.999999E+09,8.999999E+09,8.999999E+09,8.999999E+09]];
    LOCAL CONST Robtarget Tr_meulage_motif_1_231 := [[-31.666615234375,61.138640625,40.15245703125],[0.360190468749215,-0.346276211408762,0.600337290207395,-0.624460366733596],[0,0,0,0],[8.999999E+09,8.999999E+09,8.999999E+09,8.999999E+09,8.999999E+09,8.999999E+09]];
    LOCAL CONST Robtarget Tr_meulage_motif_1_232 := [[-32.1433984375,60.25962109375,40.15244140625],[0.360190468749215,-0.346276211408762,0.600337290207395,-0.624460366733596],[0,0,0,0],[8.999999E+09,8.999999E+09,8.999999E+09,8.999999E+09,8.999999E+09,8.999999E+09]];
    LOCAL CONST Robtarget Tr_meulage_motif_1_233 := [[-32.620181640625,59.3806015625,40.15242578125],[0.360190468749215,-0.346276211408762,0.600337290207395,-0.624460366733596],[0,0,0,0],[8.999999E+09,8.999999E+09,8.999999E+09,8.999999E+09,8.999999E+09,8.999999E+09]];
    LOCAL CONST Robtarget Tr_meulage_motif_1_234 := [[-33.09696484375,58.501578125,40.15241015625],[0.360190468749215,-0.346276211408762,0.600337290207395,-0.624460366733596],[0,0,0,0],[8.999999E+09,8.999999E+09,8.999999E+09,8.999999E+09,8.999999E+09,8.999999E+09]];
    LOCAL CONST Robtarget Tr_meulage_motif_1_235 := [[-33.57374609375,57.62255859375,40.15239453125],[0.360190468749215,-0.346276211408762,0.600337290207395,-0.624460366733596],[0,0,0,0],[8.999999E+09,8.999999E+09,8.999999E+09,8.999999E+09,8.999999E+09,8.999999E+09]];
    LOCAL CONST Robtarget Tr_meulage_motif_1_236 := [[-34.05053125,56.74353515625,40.15237890625],[0.360190468749215,-0.346276211408762,0.600337290207395,-0.624460366733596],[0,0,0,0],[8.999999E+09,8.999999E+09,8.999999E+09,8.999999E+09,8.999999E+09,8.999999E+09]];
    LOCAL CONST Robtarget Tr_meulage_motif_1_237 := [[-34.525171875,55.87181640625,40.04176171875],[0.360190468749215,-0.346276211408762,0.600337290207395,-0.624460366733596],[0,0,0,0],[8.999999E+09,8.999999E+09,8.999999E+09,8.999999E+09,8.999999E+09,8.999999E+09]];
    LOCAL CONST Robtarget Tr_meulage_motif_1_238 := [[-34.9791328125,55.04128515625,39.83058203125],[0.360190468749215,-0.346276211408762,0.600337290207395,-0.624460366733596],[0,0,0,0],[8.999999E+09,8.999999E+09,8.999999E+09,8.999999E+09,8.999999E+09,8.999999E+09]];
    LOCAL CONST Robtarget Tr_meulage_motif_1_239 := [[-35.3891484375,54.29360546875,39.55876953125],[0.360190468749215,-0.346276211408762,0.600337290207395,-0.624460366733596],[0,0,0,0],[8.999999E+09,8.999999E+09,8.999999E+09,8.999999E+09,8.999999E+09,8.999999E+09]];
    LOCAL CONST Robtarget Tr_meulage_motif_1_240 := [[-35.73224609375,53.67028515625,39.2546484375],[0.360190468749215,-0.346276211408762,0.600337290207395,-0.624460366733596],[0,0,0,0],[8.999999E+09,8.999999E+09,8.999999E+09,8.999999E+09,8.999999E+09,8.999999E+09]];
    LOCAL CONST Robtarget Tr_meulage_motif_1_241 := [[-36.2338828125,52.76554296875,38.592171875],[0.360190468749215,-0.346276211408762,0.600337290207395,-0.624460366733596],[0,0,0,0],[8.999999E+09,8.999999E+09,8.999999E+09,8.999999E+09,8.999999E+09,8.999999E+09]];
    LOCAL CONST Robtarget Tr_meulage_motif_1_242 := [[-36.633390625,52.05750390625,37.6524765625],[0.360190468749215,-0.346276211408762,0.600337290207395,-0.624460366733596],[0,0,0,0],[8.999999E+09,8.999999E+09,8.999999E+09,8.999999E+09,8.999999E+09,8.999999E+09]];
    LOCAL CONST Robtarget Tr_meulage_motif_1_243 := [[-36.81408984375,51.75459375,36.65621484375],[0.360190468749215,-0.346276211408762,0.600337290207395,-0.624460366733596],[0,0,0,0],[8.999999E+09,8.999999E+09,8.999999E+09,8.999999E+09,8.999999E+09,8.999999E+09]];
    LOCAL CONST Robtarget Tr_meulage_motif_1_244 := [[-36.8070390625,51.784515625,36.0987265625],[0.360190468749215,-0.346276211408762,0.600337290207395,-0.624460366733596],[0,0,0,0],[8.999999E+09,8.999999E+09,8.999999E+09,8.999999E+09,8.999999E+09,8.999999E+09]];
    LOCAL CONST Robtarget Tr_meulage_motif_1_245 := [[-36.81440625,51.78361328125,35.68086328125],[0.360190468749215,-0.346276211408762,0.600337290207395,-0.624460366733596],[0,0,0,0],[8.999999E+09,8.999999E+09,8.999999E+09,8.999999E+09,8.999999E+09,8.999999E+09]];
    LOCAL CONST Robtarget Tr_meulage_motif_1_246 := [[-36.6540546875,52.10865625,34.71164453125],[0.360190468749215,-0.346276211408762,0.600337290207395,-0.624460366733596],[0,0,0,0],[8.999999E+09,8.999999E+09,8.999999E+09,8.999999E+09,8.999999E+09,8.999999E+09]];
    LOCAL CONST Robtarget Tr_meulage_motif_1_247 := [[-36.27383203125,52.83749609375,33.7940625],[0.360190468749215,-0.346276211408762,0.600337290207395,-0.624460366733596],[0,0,0,0],[8.999999E+09,8.999999E+09,8.999999E+09,8.999999E+09,8.999999E+09,8.999999E+09]];
    LOCAL CONST Robtarget Tr_meulage_motif_1_248 := [[-35.98733984375,53.37851953125,33.3712265625],[0.360190468749215,-0.346276211408762,0.600337290207395,-0.624460366733596],[0,0,0,0],[8.999999E+09,8.999999E+09,8.999999E+09,8.999999E+09,8.999999E+09,8.999999E+09]];
    LOCAL CONST Robtarget Tr_meulage_motif_1_249 := [[-35.45516796875,54.37575390625,32.84084765625],[0.360190468749215,-0.346276211408762,0.600337290207395,-0.624460366733596],[0,0,0,0],[8.999999E+09,8.999999E+09,8.999999E+09,8.999999E+09,8.999999E+09,8.999999E+09]];
    LOCAL CONST Robtarget Tr_meulage_motif_1_250 := [[-35.05562890625,55.12037890625,32.576779296875],[0.360190468749215,-0.346276211408762,0.600337290207395,-0.624460366733596],[0,0,0,0],[8.999999E+09,8.999999E+09,8.999999E+09,8.999999E+09,8.999999E+09,8.999999E+09]];
    LOCAL CONST Robtarget Tr_meulage_motif_1_251 := [[-34.6138671875,55.9410390625,32.37233203125],[0.360190468749215,-0.346276211408762,0.600337290207395,-0.624460366733596],[0,0,0,0],[8.999999E+09,8.999999E+09,8.999999E+09,8.999999E+09,8.999999E+09,8.999999E+09]];
    LOCAL CONST Robtarget Tr_meulage_motif_1_252 := [[-34.14725390625,56.80460546875,32.2638125],[0.360190468749215,-0.346276211408762,0.600337290207395,-0.624460366733596],[0,0,0,0],[8.999999E+09,8.999999E+09,8.999999E+09,8.999999E+09,8.999999E+09,8.999999E+09]];
    LOCAL CONST Robtarget Tr_meulage_motif_1_253 := [[-33.675421875,57.6778515625,32.15323046875],[0.360190468749215,-0.346276211408762,0.600337290207395,-0.624460366733596],[0,0,0,0],[8.999999E+09,8.999999E+09,8.999999E+09,8.999999E+09,8.999999E+09,8.999999E+09]];
    LOCAL CONST Robtarget Tr_meulage_motif_1_254 := [[-33.198640625,58.556875,32.15324609375],[0.360190468749215,-0.346276211408762,0.600337290207395,-0.624460366733596],[0,0,0,0],[8.999999E+09,8.999999E+09,8.999999E+09,8.999999E+09,8.999999E+09,8.999999E+09]];
    LOCAL CONST Robtarget Tr_meulage_motif_1_255 := [[-32.72185546875,59.43589453125,32.15326171875],[0.360190468749215,-0.346276211408762,0.600337290207395,-0.624460366733596],[0,0,0,0],[8.999999E+09,8.999999E+09,8.999999E+09,8.999999E+09,8.999999E+09,8.999999E+09]];
    LOCAL CONST Robtarget Tr_meulage_motif_1_256 := [[-32.245072265625,60.3149140625,32.153279296875],[0.360190468749215,-0.346276211408762,0.600337290207395,-0.624460366733596],[0,0,0,0],[8.999999E+09,8.999999E+09,8.999999E+09,8.999999E+09,8.999999E+09,8.999999E+09]];
    LOCAL CONST Robtarget Tr_meulage_motif_1_257 := [[-31.7682890625,61.1939375,32.153294921875],[0.360190468749215,-0.346276211408762,0.600337290207395,-0.624460366733596],[0,0,0,0],[8.999999E+09,8.999999E+09,8.999999E+09,8.999999E+09,8.999999E+09,8.999999E+09]];
    LOCAL CONST Robtarget Tr_meulage_motif_1_258 := [[-31.291505859375,62.07295703125,32.153310546875],[0.360190468749215,-0.346276211408762,0.600337290207395,-0.624460366733596],[0,0,0,0],[8.999999E+09,8.999999E+09,8.999999E+09,8.999999E+09,8.999999E+09,8.999999E+09]];
    LOCAL CONST Robtarget Tr_meulage_motif_1_259 := [[-30.81472265625,62.9519765625,32.153326171875],[0.360190468749215,-0.346276211408762,0.600337290207395,-0.624460366733596],[0,0,0,0],[8.999999E+09,8.999999E+09,8.999999E+09,8.999999E+09,8.999999E+09,8.999999E+09]];
    LOCAL CONST Robtarget Tr_meulage_motif_1_260 := [[-30.337939453125,63.831,32.15334375],[0.360190468749215,-0.346276211408762,0.600337290207395,-0.624460366733596],[0,0,0,0],[8.999999E+09,8.999999E+09,8.999999E+09,8.999999E+09,8.999999E+09,8.999999E+09]];
    LOCAL CONST Robtarget Tr_meulage_motif_1_261 := [[-29.861158203125,64.71001953125,32.153359375],[0.360190468749215,-0.346276211408762,0.600337290207395,-0.624460366733596],[0,0,0,0],[8.999999E+09,8.999999E+09,8.999999E+09,8.999999E+09,8.999999E+09,8.999999E+09]];
    LOCAL CONST Robtarget Tr_meulage_motif_1_262 := [[-29.384375,65.5890390625,32.153375],[0.360190468749215,-0.346276211408762,0.600337290207395,-0.624460366733596],[0,0,0,0],[8.999999E+09,8.999999E+09,8.999999E+09,8.999999E+09,8.999999E+09,8.999999E+09]];
    LOCAL CONST Robtarget Tr_meulage_motif_1_263 := [[-28.907591796875,66.4680625,32.153390625],[0.360190468749215,-0.346276211408762,0.600337290207395,-0.624460366733596],[0,0,0,0],[8.999999E+09,8.999999E+09,8.999999E+09,8.999999E+09,8.999999E+09,8.999999E+09]];
    LOCAL CONST Robtarget Tr_meulage_motif_1_264 := [[-28.43080859375,67.3470859375,32.15340625],[0.360190468749215,-0.346276211408762,0.600337290207395,-0.624460366733596],[0,0,0,0],[8.999999E+09,8.999999E+09,8.999999E+09,8.999999E+09,8.999999E+09,8.999999E+09]];
    LOCAL CONST Robtarget Tr_meulage_motif_1_265 := [[-27.954025390625,68.2261015625,32.153423828125],[0.360190468749215,-0.346276211408762,0.600337290207395,-0.624460366733596],[0,0,0,0],[8.999999E+09,8.999999E+09,8.999999E+09,8.999999E+09,8.999999E+09,8.999999E+09]];
    LOCAL CONST Robtarget Tr_meulage_motif_1_266 := [[-27.4772421875,69.105125,32.153439453125],[0.360190468749215,-0.346276211408762,0.600337290207395,-0.624460366733596],[0,0,0,0],[8.999999E+09,8.999999E+09,8.999999E+09,8.999999E+09,8.999999E+09,8.999999E+09]];
    LOCAL CONST Robtarget Tr_meulage_motif_1_267 := [[-27.000458984375,69.9841484375,32.153455078125],[0.360190468749215,-0.346276211408762,0.600337290207395,-0.624460366733596],[0,0,0,0],[8.999999E+09,8.999999E+09,8.999999E+09,8.999999E+09,8.999999E+09,8.999999E+09]];
    LOCAL CONST Robtarget Tr_meulage_motif_1_268 := [[-26.52367578125,70.8631640625,32.153470703125],[0.360190468749215,-0.346276211408762,0.600337290207395,-0.624460366733596],[0,0,0,0],[8.999999E+09,8.999999E+09,8.999999E+09,8.999999E+09,8.999999E+09,8.999999E+09]];
    LOCAL CONST Robtarget Tr_meulage_motif_1_269 := [[-26.046892578125,71.7421875,32.15348828125],[0.360190468749215,-0.346276211408762,0.600337290207395,-0.624460366733596],[0,0,0,0],[8.999999E+09,8.999999E+09,8.999999E+09,8.999999E+09,8.999999E+09,8.999999E+09]];
    LOCAL CONST Robtarget Tr_meulage_motif_1_270 := [[-25.570109375,72.6212109375,32.15350390625],[0.360190468749215,-0.346276211408762,0.600337290207395,-0.624460366733596],[0,0,0,0],[8.999999E+09,8.999999E+09,8.999999E+09,8.999999E+09,8.999999E+09,8.999999E+09]];
    LOCAL CONST Robtarget Tr_meulage_motif_1_271 := [[-25.093326171875,73.5002265625,32.15351953125],[0.360190468749215,-0.346276211408762,0.600337290207395,-0.624460366733596],[0,0,0,0],[8.999999E+09,8.999999E+09,8.999999E+09,8.999999E+09,8.999999E+09,8.999999E+09]];
    LOCAL CONST Robtarget Tr_meulage_motif_1_272 := [[-24.61654296875,74.37925,32.15353515625],[0.360190468749215,-0.346276211408762,0.600337290207395,-0.624460366733596],[0,0,0,0],[8.999999E+09,8.999999E+09,8.999999E+09,8.999999E+09,8.999999E+09,8.999999E+09]];
    LOCAL CONST Robtarget Tr_meulage_motif_1_273 := [[-24.139759765625,75.2582734375,32.15355078125],[0.360190468749215,-0.346276211408762,0.600337290207395,-0.624460366733596],[0,0,0,0],[8.999999E+09,8.999999E+09,8.999999E+09,8.999999E+09,8.999999E+09,8.999999E+09]];
    LOCAL CONST Robtarget Tr_meulage_motif_1_274 := [[-23.6629765625,76.137296875,32.153568359375],[0.360190468749215,-0.346276211408762,0.600337290207395,-0.624460366733596],[0,0,0,0],[8.999999E+09,8.999999E+09,8.999999E+09,8.999999E+09,8.999999E+09,8.999999E+09]];
    LOCAL CONST Robtarget Tr_meulage_motif_1_275 := [[-23.186193359375,77.0163125,32.153583984375],[0.360190468749215,-0.346276211408762,0.600337290207395,-0.624460366733596],[0,0,0,0],[8.999999E+09,8.999999E+09,8.999999E+09,8.999999E+09,8.999999E+09,8.999999E+09]];
    LOCAL CONST Robtarget Tr_meulage_motif_1_276 := [[-22.709412109375,77.8953359375,32.153599609375],[0.360190468749215,-0.346276211408762,0.600337290207395,-0.624460366733596],[0,0,0,0],[8.999999E+09,8.999999E+09,8.999999E+09,8.999999E+09,8.999999E+09,8.999999E+09]];
    LOCAL CONST Robtarget Tr_meulage_motif_1_277 := [[-22.23262890625,78.774359375,32.153615234375],[0.360190468749215,-0.346276211408762,0.600337290207395,-0.624460366733596],[0,0,0,0],[8.999999E+09,8.999999E+09,8.999999E+09,8.999999E+09,8.999999E+09,8.999999E+09]];
    LOCAL CONST Robtarget Tr_meulage_motif_1_278 := [[-21.755845703125,79.653375,32.1536328125],[0.360190468749215,-0.346276211408762,0.600337290207395,-0.624460366733596],[0,0,0,0],[8.999999E+09,8.999999E+09,8.999999E+09,8.999999E+09,8.999999E+09,8.999999E+09]];
    LOCAL CONST Robtarget Tr_meulage_motif_1_279 := [[-21.2790625,80.5323984375,32.1536484375],[0.360190468749215,-0.346276211408762,0.600337290207395,-0.624460366733596],[0,0,0,0],[8.999999E+09,8.999999E+09,8.999999E+09,8.999999E+09,8.999999E+09,8.999999E+09]];
    LOCAL CONST Robtarget Tr_meulage_motif_1_280 := [[-20.802279296875,81.411421875,32.1536640625],[0.360190468749215,-0.346276211408762,0.600337290207395,-0.624460366733596],[0,0,0,0],[8.999999E+09,8.999999E+09,8.999999E+09,8.999999E+09,8.999999E+09,8.999999E+09]];
    LOCAL CONST Robtarget Tr_meulage_motif_1_281 := [[-20.32549609375,82.2904375,32.1536796875],[0.360190468749215,-0.346276211408762,0.600337290207395,-0.624460366733596],[0,0,0,0],[8.999999E+09,8.999999E+09,8.999999E+09,8.999999E+09,8.999999E+09,8.999999E+09]];
    LOCAL CONST Robtarget Tr_meulage_motif_1_282 := [[-19.848712890625,83.1694609375,32.1536953125],[0.360190468749215,-0.346276211408762,0.600337290207395,-0.624460366733596],[0,0,0,0],[8.999999E+09,8.999999E+09,8.999999E+09,8.999999E+09,8.999999E+09,8.999999E+09]];
    LOCAL CONST Robtarget Tr_meulage_motif_1_283 := [[-19.3719296875,84.048484375,32.153712890625],[0.360190468749215,-0.346276211408762,0.600337290207395,-0.624460366733596],[0,0,0,0],[8.999999E+09,8.999999E+09,8.999999E+09,8.999999E+09,8.999999E+09,8.999999E+09]];
    LOCAL CONST Robtarget Tr_meulage_motif_1_284 := [[-18.895146484375,84.9275,32.153728515625],[0.360190468749215,-0.346276211408762,0.600337290207395,-0.624460366733596],[0,0,0,0],[8.999999E+09,8.999999E+09,8.999999E+09,8.999999E+09,8.999999E+09,8.999999E+09]];
    LOCAL CONST Robtarget Tr_meulage_motif_1_285 := [[-18.41836328125,85.8065234375,32.153744140625],[0.360190468749215,-0.346276211408762,0.600337290207395,-0.624460366733596],[0,0,0,0],[8.999999E+09,8.999999E+09,8.999999E+09,8.999999E+09,8.999999E+09,8.999999E+09]];
    LOCAL CONST Robtarget Tr_meulage_motif_1_286 := [[-17.941580078125,86.685546875,32.153759765625],[0.360190468749215,-0.346276211408762,0.600337290207395,-0.624460366733596],[0,0,0,0],[8.999999E+09,8.999999E+09,8.999999E+09,8.999999E+09,8.999999E+09,8.999999E+09]];
    LOCAL CONST Robtarget Tr_meulage_motif_1_287 := [[-17.464796875,87.5645625,32.15377734375],[0.360190468749215,-0.346276211408762,0.600337290207395,-0.624460366733596],[0,0,0,0],[8.999999E+09,8.999999E+09,8.999999E+09,8.999999E+09,8.999999E+09,8.999999E+09]];
    LOCAL CONST Robtarget Tr_meulage_motif_1_288 := [[-16.988013671875,88.4435859375,32.15379296875],[0.360190468749215,-0.346276211408762,0.600337290207395,-0.624460366733596],[0,0,0,0],[8.999999E+09,8.999999E+09,8.999999E+09,8.999999E+09,8.999999E+09,8.999999E+09]];
    LOCAL CONST Robtarget Tr_meulage_motif_1_289 := [[-16.51123046875,89.322609375,32.15380859375],[0.360190468749215,-0.346276211408762,0.600337290207395,-0.624460366733596],[0,0,0,0],[8.999999E+09,8.999999E+09,8.999999E+09,8.999999E+09,8.999999E+09,8.999999E+09]];
    LOCAL CONST Robtarget Tr_meulage_motif_1_290 := [[-16.0344482421875,90.2016328125,32.15382421875],[0.360190468749215,-0.346276211408762,0.600337290207395,-0.624460366733596],[0,0,0,0],[8.999999E+09,8.999999E+09,8.999999E+09,8.999999E+09,8.999999E+09,8.999999E+09]];
    LOCAL CONST Robtarget Tr_meulage_motif_1_291 := [[-15.5576650390625,91.0806484375,32.15383984375],[0.360190468749215,-0.346276211408762,0.600337290207395,-0.624460366733596],[0,0,0,0],[8.999999E+09,8.999999E+09,8.999999E+09,8.999999E+09,8.999999E+09,8.999999E+09]];
    LOCAL CONST Robtarget Tr_meulage_motif_1_292 := [[-15.0808818359375,91.959671875,32.153857421875],[0.360190468749215,-0.346276211408762,0.600337290207395,-0.624460366733596],[0,0,0,0],[8.999999E+09,8.999999E+09,8.999999E+09,8.999999E+09,8.999999E+09,8.999999E+09]];
    LOCAL CONST Robtarget Tr_meulage_motif_1_293 := [[-14.6040986328125,92.8386953125,32.153873046875],[0.360190468749215,-0.346276211408762,0.600337290207395,-0.624460366733596],[0,0,0,0],[8.999999E+09,8.999999E+09,8.999999E+09,8.999999E+09,8.999999E+09,8.999999E+09]];
    LOCAL CONST Robtarget Tr_meulage_motif_1_294 := [[-14.1273154296875,93.7177109375,32.153888671875],[0.360190468749215,-0.346276211408762,0.600337290207395,-0.624460366733596],[0,0,0,0],[8.999999E+09,8.999999E+09,8.999999E+09,8.999999E+09,8.999999E+09,8.999999E+09]];

